LIN {X 0,Y 439.406,Z 545.749,A -85,B 0,C 180,E1 -8966.874,E2 -8966.874} C_VEL
LIN {X 0,Y 444.301,Z 559.149,A -85,B 0,C 180,E1 -8967.337,E2 -8967.337} C_VEL
LIN {X 0,Y 445.02,Z 561.087,A -85,B 0,C 180,E1 -8967.401,E2 -8967.401} C_VEL
LIN {X 0,Y 444.548,Z 605.152,A -85,B 0,C 180,E1 -8968.2,E2 -8968.2} C_VEL
LIN {X 0,Y 444.368,Z 618.583,A -85,B 0,C 180,E1 -8968.612,E2 -8968.612} C_VEL
LIN {X 0,Y 444.074,Z 631.835,A -85,B 0,C 180,E1 -8969.192,E2 -8969.192} C_VEL
LIN {X 0,Y 443.603,Z 644.701,A -85,B 0,C 180,E1 -8969.932,E2 -8969.932} C_VEL
LIN {X 0,Y 443.053,Z 657.633,A -85,B 0,C 180,E1 -8970.889,E2 -8970.889} C_VEL
LIN {X 0,Y 442.359,Z 670.207,A -85,B 0,C 180,E1 -8972.052,E2 -8972.052} C_VEL
LIN {X 0,Y 441.738,Z 680.558,A -85,B 0,C 180,E1 -8973.223,E2 -8973.223} C_VEL
LIN {X 0,Y 441.181,Z 690.099,A -85,B 0,C 180,E1 -8974.526,E2 -8974.526} C_VEL
LIN {X 0,Y 440.602,Z 699.018,A -85,B 0,C 180,E1 -8976,E2 -8976} C_VEL
LIN {X 0,Y 440.165,Z 706.273,A -85,B 0,C 180,E1 -8977.468,E2 -8977.468} C_VEL
LIN {X 0,Y 439.771,Z 712.189,A -85,B 0,C 180,E1 -8978.926,E2 -8978.926} C_VEL
LIN {X 0,Y 439.514,Z 717.633,A -85,B 0,C 180,E1 -8980.634,E2 -8980.634} C_VEL
LIN {X 0,Y 439.268,Z 721.644,A -85,B 0,C 180,E1 -8982.303,E2 -8982.303} C_VEL
LIN {X 0,Y 439.103,Z 724.753,A -85,B 0,C 180,E1 -8984.212,E2 -8984.212} C_VEL
LIN {X 0,Y 439.067,Z 726.387,A -85,B 0,C 180,E1 -8986.108,E2 -8986.108} C_VEL
LIN {X 0,Y 439.137,Z 726.572,A -85,B 0,C 180,E1 -8987.992,E2 -8987.992} C_VEL
LIN {X 0,Y 439.207,Z 725.332,A -85,B 0,C 180,E1 -8989.863,E2 -8989.863} C_VEL
LIN {X 0,Y 439.399,Z 722.692,A -85,B 0,C 180,E1 -8991.724,E2 -8991.724} C_VEL
LIN {X 0,Y 439.752,Z 718.586,A -85,B 0,C 180,E1 -8993.577,E2 -8993.577} C_VEL
LIN {X 0,Y 439.994,Z 714.453,A -85,B 0,C 180,E1 -8994.96,E2 -8994.96} C_VEL
LIN {X 0,Y 440.331,Z 709.35,A -85,B 0,C 180,E1 -8996.34,E2 -8996.34} C_VEL
LIN {X 0,Y 440.85,Z 701.986,A -85,B 0,C 180,E1 -8997.945,E2 -8997.945} C_VEL
LIN {X 0,Y 441.381,Z 694.239,A -85,B 0,C 180,E1 -8999.316,E2 -8999.316} C_VEL
LIN {X 0,Y 442.094,Z 684.837,A -85,B 0,C 180,E1 -9000.684,E2 -9000.684} C_VEL
LIN {X 0,Y 442.669,Z 674.365,A -85,B 0,C 180,E1 -9001.934,E2 -9001.934} C_VEL
LIN {X 0,Y 443.376,Z 662.58,A -85,B 0,C 180,E1 -9003.067,E2 -9003.067} C_VEL
LIN {X 0,Y 443.967,Z 650.958,A -85,B 0,C 180,E1 -9003.972,E2 -9003.972} C_VEL
LIN {X 0,Y 444.369,Z 638.23,A -85,B 0,C 180,E1 -9004.763,E2 -9004.763} C_VEL
LIN {X 0,Y 444.691,Z 624.706,A -85,B 0,C 180,E1 -9005.398,E2 -9005.398} C_VEL
LIN {X 0,Y 444.834,Z 611.284,A -85,B 0,C 180,E1 -9005.838,E2 -9005.838} C_VEL
LIN {X 0,Y 444.826,Z 592.596,A -85,B 0,C 180,E1 -9006.208,E2 -9006.208} C_VEL
LIN {X 0,Y 445.192,Z 560.426,A -85,B 0,C 180,E1 -9006.758,E2 -9006.758} C_VEL
LIN {X 0,Y 439.624,Z 545.984,A -85,B 0,C 180,E1 -9007.305,E2 -9007.305} C_VEL
LIN {X 0,Y 439.598,Z 545.729,A -85,B 0,C 180,E1 -9007.349,E2 -9007.349} C_VEL
LIN {X 0,Y 439.465,Z 545.745,A -85,B 0,C 180,E1 -9010.132,E2 -9010.132} C_VEL
LIN {X 0,Y 439.47,Z 545.745,A -85,B 0,C 180,E1 -9012.938,E2 -9012.938} C_VEL
LIN {X 0,Y 439.444,Z 545.746,A -85,B 0,C 180,E1 -9016.349,E2 -9016.349} C_VEL
LIN {X 0,Y 439.4,Z 545.753,A -85,B 0,C 180,E1 -9019.627,E2 -9019.627} C_VEL
LIN {X 0,Y 439.363,Z 545.754,A -85,B 0,C 180,E1 -9022.576,E2 -9022.576} C_VEL
LIN {X 0,Y 439.403,Z 545.75,A -85,B 0,C 180,E1 -9025.585,E2 -9025.585} C_VEL
LIN {X 0,Y 439.423,Z 545.743,A -85,B 0,C 180,E1 -9028.674,E2 -9028.674} C_VEL
LIN {X 0,Y 439.373,Z 545.747,A -85,B 0,C 180,E1 -9031.861,E2 -9031.861} C_VEL
LIN {X 0,Y 439.397,Z 545.747,A -85,B 0,C 180,E1 -9035.157,E2 -9035.157} C_VEL
LIN {X 0,Y 439.388,Z 545.749,A -85,B 0,C 180,E1 -9038.595,E2 -9038.595} C_VEL
LIN {X 0,Y 439.388,Z 545.754,A -85,B 0,C 180,E1 -9041.258,E2 -9041.258} C_VEL
LIN {X 0,Y 439.404,Z 545.749,A -85,B 0,C 180,E1 -9044.729,E2 -9044.729} C_VEL
LIN {X 0,Y 439.395,Z 545.748,A -85,B 0,C 180,E1 -9047.796,E2 -9047.796} C_VEL
LIN {X 0,Y 439.429,Z 545.745,A -85,B 0,C 180,E1 -9050.229,E2 -9050.229} C_VEL
LIN {X 0,Y 439.385,Z 545.756,A -85,B 0,C 180,E1 -9053.715,E2 -9053.715} C_VEL
LIN {X 0,Y 439.429,Z 545.847,A -85,B 0,C 180,E1 -9054.275,E2 -9054.275} C_VEL
LIN {X 0,Y 442.842,Z 561.566,A -85,B 0,C 180,E1 -9057.615,E2 -9057.615} C_VEL
LIN {X 0,Y 443.621,Z 565.787,A -85,B 0,C 180,E1 -9058.481,E2 -9058.481} C_VEL
LIN {X 0,Y 442.616,Z 582.035,A -85,B 0,C 180,E1 -9061.553,E2 -9061.553} C_VEL
LIN {X 0,Y 441.489,Z 601.988,A -85,B 0,C 180,E1 -9065.244,E2 -9065.244} C_VEL
LIN {X 0,Y 440.582,Z 621.12,A -85,B 0,C 180,E1 -9068.722,E2 -9068.722} C_VEL
LIN {X 0,Y 439.955,Z 635.532,A -85,B 0,C 180,E1 -9071.278,E2 -9071.278} C_VEL
LIN {X 0,Y 444.537,Z 670.934,A -85,B 0,C 180,E1 -9072.213,E2 -9072.213} C_VEL
LIN {X 0,Y 443.06,Z 749.107,A -85,B 0,C 180,E1 -9073.795,E2 -9073.795} C_VEL
LIN {X 0,Y 442.451,Z 763.207,A -85,B 0,C 180,E1 -9074.275,E2 -9074.275} C_VEL
LIN {X 0,Y 441.799,Z 775.931,A -85,B 0,C 180,E1 -9074.902,E2 -9074.902} C_VEL
LIN {X 0,Y 441.003,Z 788.207,A -85,B 0,C 180,E1 -9075.7,E2 -9075.7} C_VEL
LIN {X 0,Y 440.449,Z 799.159,A -85,B 0,C 180,E1 -9076.601,E2 -9076.601} C_VEL
LIN {X 0,Y 439.972,Z 809.643,A -85,B 0,C 180,E1 -9077.664,E2 -9077.664} C_VEL
LIN {X 0,Y 439.354,Z 819.768,A -85,B 0,C 180,E1 -9078.934,E2 -9078.934} C_VEL
LIN {X 0,Y 438.991,Z 828.76,A -85,B 0,C 180,E1 -9080.323,E2 -9080.323} C_VEL
LIN {X 0,Y 438.777,Z 835.975,A -85,B 0,C 180,E1 -9081.712,E2 -9081.712} C_VEL
LIN {X 0,Y 438.666,Z 842.745,A -85,B 0,C 180,E1 -9083.377,E2 -9083.377} C_VEL
LIN {X 0,Y 438.702,Z 847.553,A -85,B 0,C 180,E1 -9084.946,E2 -9084.946} C_VEL
LIN {X 0,Y 438.764,Z 850.593,A -85,B 0,C 180,E1 -9086.327,E2 -9086.327} C_VEL
LIN {X 0,Y 438.733,Z 852.033,A -85,B 0,C 180,E1 -9087.246,E2 -9087.246} C_VEL
LIN {X 0,Y 438.734,Z 853.013,A -85,B 0,C 180,E1 -9088.165,E2 -9088.165} C_VEL
LIN {X 0,Y 438.737,Z 853.57,A -85,B 0,C 180,E1 -9089.083,E2 -9089.083} C_VEL
LIN {X 0,Y 438.937,Z 853.735,A -85,B 0,C 180,E1 -9090.001,E2 -9090.001} C_VEL
LIN {X 0,Y 438.76,Z 853.392,A -85,B 0,C 180,E1 -9090.918,E2 -9090.918} C_VEL
LIN {X 0,Y 438.781,Z 852.625,A -85,B 0,C 180,E1 -9091.836,E2 -9091.836} C_VEL
LIN {X 0,Y 438.797,Z 851.434,A -85,B 0,C 180,E1 -9092.755,E2 -9092.755} C_VEL
LIN {X 0,Y 438.851,Z 848.799,A -85,B 0,C 180,E1 -9094.133,E2 -9094.133} C_VEL
LIN {X 0,Y 438.771,Z 845.065,A -85,B 0,C 180,E1 -9095.515,E2 -9095.515} C_VEL
LIN {X 0,Y 438.821,Z 840.059,A -85,B 0,C 180,E1 -9096.929,E2 -9096.929} C_VEL
LIN {X 0,Y 438.886,Z 833.994,A -85,B 0,C 180,E1 -9098.287,E2 -9098.287} C_VEL
LIN {X 0,Y 439.014,Z 826.334,A -85,B 0,C 180,E1 -9099.677,E2 -9099.677} C_VEL
LIN {X 0,Y 439.34,Z 816.842,A -85,B 0,C 180,E1 -9101.068,E2 -9101.068} C_VEL
LIN {X 0,Y 439.854,Z 806.195,A -85,B 0,C 180,E1 -9102.331,E2 -9102.331} C_VEL
LIN {X 0,Y 440.138,Z 798.182,A -85,B 0,C 180,E1 -9103.129,E2 -9103.129} C_VEL
LIN {X 0,Y 440.575,Z 788.32,A -85,B 0,C 180,E1 -9103.962,E2 -9103.962} C_VEL
LIN {X 0,Y 441.416,Z 774.803,A -85,B 0,C 180,E1 -9104.877,E2 -9104.877} C_VEL
LIN {X 0,Y 442.071,Z 761.506,A -85,B 0,C 180,E1 -9105.562,E2 -9105.562} C_VEL
LIN {X 0,Y 442.834,Z 747.018,A -85,B 0,C 180,E1 -9106.096,E2 -9106.096} C_VEL
LIN {X 0,Y 443.169,Z 732.682,A -85,B 0,C 180,E1 -9106.438,E2 -9106.438} C_VEL
LIN {X 0,Y 444.068,Z 670.071,A -85,B 0,C 180,E1 -9107.651,E2 -9107.651} C_VEL
LIN {X 0,Y 442.737,Z 654.934,A -85,B 0,C 180,E1 -9108.032,E2 -9108.032} C_VEL
LIN {X 0,Y 440.919,Z 632.046,A -85,B 0,C 180,E1 -9108.615,E2 -9108.615} C_VEL
LIN {X 0,Y 439.683,Z 620.875,A -85,B 0,C 180,E1 -9108.948,E2 -9108.948} C_VEL
LIN {X 0,Y 439.902,Z 603.534,A -85,B 0,C 180,E1 -9111.823,E2 -9111.823} C_VEL
LIN {X 0,Y 440.157,Z 584.473,A -85,B 0,C 180,E1 -9115.033,E2 -9115.033} C_VEL
LIN {X 0,Y 440.516,Z 566.826,A -85,B 0,C 180,E1 -9118.077,E2 -9118.077} C_VEL
LIN {X 0,Y 440.777,Z 553.487,A -85,B 0,C 180,E1 -9120.446,E2 -9120.446} C_VEL
LIN {X 0,Y 439.477,Z 545.744,A -85,B 0,C 180,E1 -9121.938,E2 -9121.938} C_VEL
LIN {X 0,Y 439.399,Z 545.752,A -85,B 0,C 180,E1 -9125.341,E2 -9125.341} C_VEL
LIN {X 0,Y 439.383,Z 545.753,A -85,B 0,C 180,E1 -9128.595,E2 -9128.595} C_VEL
LIN {X 0,Y 439.393,Z 545.752,A -85,B 0,C 180,E1 -9131.257,E2 -9131.257} C_VEL
LIN {X 0,Y 439.405,Z 545.752,A -85,B 0,C 180,E1 -9134.729,E2 -9134.729} C_VEL
LIN {X 0,Y 439.401,Z 545.749,A -85,B 0,C 180,E1 -9137.796,E2 -9137.796} C_VEL
LIN {X 0,Y 439.434,Z 545.747,A -85,B 0,C 180,E1 -9140.228,E2 -9140.228} C_VEL
LIN {X 0,Y 439.378,Z 545.752,A -85,B 0,C 180,E1 -9143.713,E2 -9143.713} C_VEL
LIN {X 0,Y 439.377,Z 545.755,A -85,B 0,C 180,E1 -9147.054,E2 -9147.054} C_VEL
LIN {X 0,Y 439.387,Z 545.754,A -85,B 0,C 180,E1 -9150.274,E2 -9150.274} C_VEL
LIN {X 0,Y 439.433,Z 545.749,A -85,B 0,C 180,E1 -9153.396,E2 -9153.396} C_VEL
LIN {X 0,Y 439.392,Z 545.758,A -85,B 0,C 180,E1 -9156.429,E2 -9156.429} C_VEL
LIN {X 0,Y 439.393,Z 545.753,A -85,B 0,C 180,E1 -9159.397,E2 -9159.397} C_VEL
LIN {X 0,Y 439.407,Z 545.753,A -85,B 0,C 180,E1 -9160.374,E2 -9160.374} C_VEL
LIN {X 0,Y 440.396,Z 548.536,A -85,B 0,C 180,E1 -9160.485,E2 -9160.485} C_VEL
LIN {X 0,Y 445.662,Z 561.095,A -85,B 0,C 180,E1 -9160.997,E2 -9160.997} C_VEL
LIN {X 0,Y 446.009,Z 561.957,A -85,B 0,C 180,E1 -9161.029,E2 -9161.029} C_VEL
LIN {X 0,Y 445.994,Z 595.08,A -85,B 0,C 180,E1 -9161.61,E2 -9161.61} C_VEL
LIN {X 0,Y 446.007,Z 609.272,A -85,B 0,C 180,E1 -9162.028,E2 -9162.028} C_VEL
LIN {X 0,Y 445.804,Z 623.559,A -85,B 0,C 180,E1 -9162.629,E2 -9162.629} C_VEL
LIN {X 0,Y 445.368,Z 637.072,A -85,B 0,C 180,E1 -9163.38,E2 -9163.38} C_VEL
LIN {X 0,Y 444.838,Z 650.124,A -85,B 0,C 180,E1 -9164.302,E2 -9164.302} C_VEL
LIN {X 0,Y 444.15,Z 663.194,A -85,B 0,C 180,E1 -9165.451,E2 -9165.451} C_VEL
LIN {X 0,Y 443.548,Z 673.013,A -85,B 0,C 180,E1 -9166.484,E2 -9166.484} C_VEL
LIN {X 0,Y 442.758,Z 683.962,A -85,B 0,C 180,E1 -9167.858,E2 -9167.858} C_VEL
LIN {X 0,Y 442.052,Z 693.037,A -85,B 0,C 180,E1 -9169.233,E2 -9169.233} C_VEL
LIN {X 0,Y 441.414,Z 701.82,A -85,B 0,C 180,E1 -9170.838,E2 -9170.838} C_VEL
LIN {X 0,Y 440.947,Z 708.047,A -85,B 0,C 180,E1 -9172.213,E2 -9172.213} C_VEL
LIN {X 0,Y 440.344,Z 713.376,A -85,B 0,C 180,E1 -9173.585,E2 -9173.585} C_VEL
LIN {X 0,Y 440.027,Z 719.004,A -85,B 0,C 180,E1 -9175.419,E2 -9175.419} C_VEL
LIN {X 0,Y 439.637,Z 723.262,A -85,B 0,C 180,E1 -9177.251,E2 -9177.251} C_VEL
LIN {X 0,Y 439.42,Z 726.213,A -85,B 0,C 180,E1 -9179.083,E2 -9179.083} C_VEL
LIN {X 0,Y 439.321,Z 727.927,A -85,B 0,C 180,E1 -9180.916,E2 -9180.916} C_VEL
LIN {X 0,Y 439.331,Z 728.446,A -85,B 0,C 180,E1 -9182.75,E2 -9182.75} C_VEL
LIN {X 0,Y 439.21,Z 727.821,A -85,B 0,C 180,E1 -9184.589,E2 -9184.589} C_VEL
LIN {X 0,Y 439.375,Z 725.987,A -85,B 0,C 180,E1 -9186.428,E2 -9186.428} C_VEL
LIN {X 0,Y 439.475,Z 722.948,A -85,B 0,C 180,E1 -9188.275,E2 -9188.275} C_VEL
LIN {X 0,Y 439.667,Z 718.609,A -85,B 0,C 180,E1 -9190.127,E2 -9190.127} C_VEL
LIN {X 0,Y 439.974,Z 712.852,A -85,B 0,C 180,E1 -9191.985,E2 -9191.985} C_VEL
LIN {X 0,Y 440.486,Z 705.487,A -85,B 0,C 180,E1 -9193.846,E2 -9193.846} C_VEL
LIN {X 0,Y 441.044,Z 697.51,A -85,B 0,C 180,E1 -9195.48,E2 -9195.48} C_VEL
LIN {X 0,Y 441.581,Z 689.227,A -85,B 0,C 180,E1 -9196.901,E2 -9196.901} C_VEL
LIN {X 0,Y 442.224,Z 679.63,A -85,B 0,C 180,E1 -9198.292,E2 -9198.292} C_VEL
LIN {X 0,Y 442.965,Z 667.969,A -85,B 0,C 180,E1 -9199.703,E2 -9199.703} C_VEL
LIN {X 0,Y 443.641,Z 656.875,A -85,B 0,C 180,E1 -9200.826,E2 -9200.826} C_VEL
LIN {X 0,Y 444.248,Z 645.173,A -85,B 0,C 180,E1 -9201.824,E2 -9201.824} C_VEL
LIN {X 0,Y 444.838,Z 631.595,A -85,B 0,C 180,E1 -9202.772,E2 -9202.772} C_VEL
LIN {X 0,Y 445.415,Z 616.975,A -85,B 0,C 180,E1 -9203.573,E2 -9203.573} C_VEL
LIN {X 0,Y 445.77,Z 601.844,A -85,B 0,C 180,E1 -9204.199,E2 -9204.199} C_VEL
LIN {X 0,Y 445.907,Z 586.802,A -85,B 0,C 180,E1 -9204.635,E2 -9204.635} C_VEL
LIN {X 0,Y 445.984,Z 563.306,A -85,B 0,C 180,E1 -9205.079,E2 -9205.079} C_VEL
LIN {X 0,Y 439.464,Z 545.989,A -85,B 0,C 180,E1 -9205.687,E2 -9205.687} C_VEL
LIN {X 0,Y 439.43,Z 545.751,A -85,B 0,C 180,E1 -9205.837,E2 -9205.837} C_VEL
LIN {X 0,Y 439.419,Z 545.747,A -85,B 0,C 180,E1 -9208.673,E2 -9208.673} C_VEL
LIN {X 0,Y 439.372,Z 545.758,A -85,B 0,C 180,E1 -9212.03,E2 -9212.03} C_VEL
LIN {X 0,Y 439.395,Z 545.747,A -85,B 0,C 180,E1 -9215.34,E2 -9215.34} C_VEL
LIN {X 0,Y 439.379,Z 545.752,A -85,B 0,C 180,E1 -9218.595,E2 -9218.595} C_VEL
LIN {X 0,Y 439.389,Z 545.748,A -85,B 0,C 180,E1 -9221.256,E2 -9221.256} C_VEL
LIN {X 0,Y 439.4,Z 545.749,A -85,B 0,C 180,E1 -9224.729,E2 -9224.729} C_VEL
LIN {X 0,Y 439.396,Z 545.749,A -85,B 0,C 180,E1 -9227.795,E2 -9227.795} C_VEL
LIN {X 0,Y 439.436,Z 545.748,A -85,B 0,C 180,E1 -9230.228,E2 -9230.228} C_VEL
LIN {X 0,Y 439.376,Z 545.75,A -85,B 0,C 180,E1 -9233.712,E2 -9233.712} C_VEL
LIN {X 0,Y 439.372,Z 545.752,A -85,B 0,C 180,E1 -9237.053,E2 -9237.053} C_VEL
LIN {X 0,Y 439.382,Z 545.753,A -85,B 0,C 180,E1 -9240.274,E2 -9240.274} C_VEL
LIN {X 0,Y 439.429,Z 545.743,A -85,B 0,C 180,E1 -9243.396,E2 -9243.396} C_VEL
LIN {X 0,Y 439.387,Z 545.753,A -85,B 0,C 180,E1 -9246.429,E2 -9246.429} C_VEL
LIN {X 0,Y 439.388,Z 545.749,A -85,B 0,C 180,E1 -9249.397,E2 -9249.397} C_VEL
LIN {X 0,Y 439.43,Z 545.745,A -85,B 0,C 180,E1 -9252.309,E2 -9252.309} C_VEL
LIN {X 0,Y 439.447,Z 545.745,A -85,B 0,C 180,E1 -9255.173,E2 -9255.173} C_VEL
LIN {X 0,Y 439.482,Z 545.736,A -85,B 0,C 180,E1 -9258.001,E2 -9258.001} C_VEL
LIN {X 0,Y 439.528,Z 545.731,A -85,B 0,C 180,E1 -9261.547,E2 -9261.547} C_VEL
LIN {X 0,Y 438.908,Z 545.81,A -85,B 0,C 180,E1 -9262.313,E2 -9262.313} C_VEL
LIN {X 0,Y 436.034,Z 546.171,A -85,B 0,C 180,E1 -9263.556,E2 -9263.556} C_VEL
LIN {X 0,Y 433.558,Z 546.481,A -85,B 0,C 180,E1 -9264.559,E2 -9264.559} C_VEL
LIN {X 0,Y 432.477,Z 546.614,A -85,B 0,C 180,E1 -9265.334,E2 -9265.334} C_VEL
LIN {X 0,Y 432.382,Z 546.622,A -85,B 0,C 180,E1 -9265.597,E2 -9265.597} C_VEL
LIN {X 0,Y 432.604,Z 546.593,A -85,B 0,C 180,E1 -9268.137,E2 -9268.137} C_VEL
LIN {X 0,Y 432.732,Z 546.577,A -85,B 0,C 180,E1 -9269.999,E2 -9269.999} C_VEL
LIN {X 0,Y 432.604,Z 546.596,A -85,B 0,C 180,E1 -9272.793,E2 -9272.793} C_VEL
LIN {X 0,Y 432.562,Z 546.599,A -85,B 0,C 180,E1 -9276.53,E2 -9276.53} C_VEL
LIN {X 0,Y 432.441,Z 546.621,A -85,B 0,C 180,E1 -9279.353,E2 -9279.353} C_VEL
LIN {X 0,Y 432.442,Z 546.615,A -85,B 0,C 180,E1 -9282.812,E2 -9282.812} C_VEL
LIN {X 0,Y 432.409,Z 546.617,A -85,B 0,C 180,E1 -9286.479,E2 -9286.479} C_VEL
LIN {X 0,Y 432.335,Z 546.629,A -85,B 0,C 180,E1 -9289.96,E2 -9289.96} C_VEL
LIN {X 0,Y 432.316,Z 546.63,A -85,B 0,C 180,E1 -9292.964,E2 -9292.964} C_VEL
LIN {X 0,Y 432.361,Z 546.626,A -85,B 0,C 180,E1 -9296.032,E2 -9296.032} C_VEL
LIN {X 0,Y 432.348,Z 546.627,A -85,B 0,C 180,E1 -9299.186,E2 -9299.186} C_VEL
LIN {X 0,Y 432.327,Z 546.629,A -85,B 0,C 180,E1 -9302.294,E2 -9302.294} C_VEL
LIN {X 0,Y 432.336,Z 546.627,A -85,B 0,C 180,E1 -9304.677,E2 -9304.677} C_VEL
LIN {X 0,Y 432.346,Z 546.629,A -85,B 0,C 180,E1 -9308.148,E2 -9308.148} C_VEL
LIN {X 0,Y 432.361,Z 546.627,A -85,B 0,C 180,E1 -9311.607,E2 -9311.607} C_VEL
LIN {X 0,Y 432.332,Z 546.63,A -85,B 0,C 180,E1 -9314.347,E2 -9314.347} C_VEL
LIN {X 0,Y 432.36,Z 546.623,A -85,B 0,C 180,E1 -9317.009,E2 -9317.009} C_VEL
LIN {X 0,Y 432.355,Z 546.629,A -85,B 0,C 180,E1 -9319.816,E2 -9319.816} C_VEL
LIN {X 0,Y 432.312,Z 546.629,A -85,B 0,C 180,E1 -9323.023,E2 -9323.023} C_VEL
LIN {X 0,Y 432.371,Z 546.626,A -85,B 0,C 180,E1 -9326.535,E2 -9326.535} C_VEL
LIN {X 0,Y 432.415,Z 546.866,A -85,B 0,C 180,E1 -9326.623,E2 -9326.623} C_VEL
LIN {X 0,Y 438.178,Z 562.466,A -85,B 0,C 180,E1 -9327.152,E2 -9327.152} C_VEL
LIN {X 0,Y 437.739,Z 605.294,A -85,B 0,C 180,E1 -9327.943,E2 -9327.943} C_VEL
LIN {X 0,Y 437.568,Z 619.263,A -85,B 0,C 180,E1 -9328.372,E2 -9328.372} C_VEL
LIN {X 0,Y 437.269,Z 632.342,A -85,B 0,C 180,E1 -9328.948,E2 -9328.948} C_VEL
LIN {X 0,Y 436.792,Z 645.03,A -85,B 0,C 180,E1 -9329.681,E2 -9329.681} C_VEL
LIN {X 0,Y 436.274,Z 657.064,A -85,B 0,C 180,E1 -9330.562,E2 -9330.562} C_VEL
LIN {X 0,Y 435.648,Z 668.401,A -85,B 0,C 180,E1 -9331.582,E2 -9331.582} C_VEL
LIN {X 0,Y 434.942,Z 679.636,A -85,B 0,C 180,E1 -9332.821,E2 -9332.821} C_VEL
LIN {X 0,Y 434.319,Z 689.176,A -85,B 0,C 180,E1 -9334.094,E2 -9334.094} C_VEL
LIN {X 0,Y 433.754,Z 698.457,A -85,B 0,C 180,E1 -9335.596,E2 -9335.596} C_VEL
LIN {X 0,Y 433.257,Z 706.021,A -85,B 0,C 180,E1 -9337.089,E2 -9337.089} C_VEL
LIN {X 0,Y 432.845,Z 712.177,A -85,B 0,C 180,E1 -9338.573,E2 -9338.573} C_VEL
LIN {X 0,Y 432.568,Z 717.133,A -85,B 0,C 180,E1 -9340.051,E2 -9340.051} C_VEL
LIN {X 0,Y 432.356,Z 721.035,A -85,B 0,C 180,E1 -9341.52,E2 -9341.52} C_VEL
LIN {X 0,Y 432.158,Z 723.999,A -85,B 0,C 180,E1 -9342.979,E2 -9342.979} C_VEL
LIN {X 0,Y 432.037,Z 726.542,A -85,B 0,C 180,E1 -9344.914,E2 -9344.914} C_VEL
LIN {X 0,Y 432.078,Z 727.631,A -85,B 0,C 180,E1 -9346.838,E2 -9346.838} C_VEL
LIN {X 0,Y 432.111,Z 727.328,A -85,B 0,C 180,E1 -9348.746,E2 -9348.746} C_VEL
LIN {X 0,Y 432.279,Z 725.572,A -85,B 0,C 180,E1 -9350.644,E2 -9350.644} C_VEL
LIN {X 0,Y 432.549,Z 722.374,A -85,B 0,C 180,E1 -9352.532,E2 -9352.532} C_VEL
LIN {X 0,Y 432.895,Z 717.686,A -85,B 0,C 180,E1 -9354.41,E2 -9354.41} C_VEL
LIN {X 0,Y 433.213,Z 713.068,A -85,B 0,C 180,E1 -9355.814,E2 -9355.814} C_VEL
LIN {X 0,Y 433.767,Z 706.35,A -85,B 0,C 180,E1 -9357.447,E2 -9357.447} C_VEL
LIN {X 0,Y 434.253,Z 699.278,A -85,B 0,C 180,E1 -9358.841,E2 -9358.841} C_VEL
LIN {X 0,Y 434.957,Z 690.7,A -85,B 0,C 180,E1 -9360.232,E2 -9360.232} C_VEL
LIN {X 0,Y 435.498,Z 682.189,A -85,B 0,C 180,E1 -9361.387,E2 -9361.387} C_VEL
LIN {X 0,Y 436.155,Z 672.098,A -85,B 0,C 180,E1 -9362.53,E2 -9362.53} C_VEL
LIN {X 0,Y 436.802,Z 660.849,A -85,B 0,C 180,E1 -9363.575,E2 -9363.575} C_VEL
LIN {X 0,Y 437.413,Z 648.462,A -85,B 0,C 180,E1 -9364.493,E2 -9364.493} C_VEL
LIN {X 0,Y 437.802,Z 635.629,A -85,B 0,C 180,E1 -9365.239,E2 -9365.239} C_VEL
LIN {X 0,Y 438.099,Z 621.765,A -85,B 0,C 180,E1 -9365.836,E2 -9365.836} C_VEL
LIN {X 0,Y 438.132,Z 608.616,A -85,B 0,C 180,E1 -9366.225,E2 -9366.225} C_VEL
LIN {X 0,Y 438.569,Z 562.004,A -85,B 0,C 180,E1 -9367.058,E2 -9367.058} C_VEL
LIN {X 0,Y 432.674,Z 547.122,A -85,B 0,C 180,E1 -9367.662,E2 -9367.662} C_VEL
LIN {X 0,Y 432.56,Z 546.606,A -85,B 0,C 180,E1 -9367.698,E2 -9367.698} C_VEL
LIN {X 0,Y 432.405,Z 546.625,A -85,B 0,C 180,E1 -9371.247,E2 -9371.247} C_VEL
LIN {X 0,Y 432.428,Z 546.624,A -85,B 0,C 180,E1 -9373.152,E2 -9373.152} C_VEL
LIN {X 0,Y 432.409,Z 546.622,A -85,B 0,C 180,E1 -9376.48,E2 -9376.48} C_VEL
LIN {X 0,Y 432.336,Z 546.633,A -85,B 0,C 180,E1 -9379.961,E2 -9379.961} C_VEL
LIN {X 0,Y 432.317,Z 546.634,A -85,B 0,C 180,E1 -9382.965,E2 -9382.965} C_VEL
LIN {X 0,Y 432.362,Z 546.625,A -85,B 0,C 180,E1 -9386.033,E2 -9386.033} C_VEL
LIN {X 0,Y 432.35,Z 546.629,A -85,B 0,C 180,E1 -9389.187,E2 -9389.187} C_VEL
LIN {X 0,Y 432.323,Z 546.623,A -85,B 0,C 180,E1 -9392.294,E2 -9392.294} C_VEL
LIN {X 0,Y 432.338,Z 546.624,A -85,B 0,C 180,E1 -9394.678,E2 -9394.678} C_VEL
LIN {X 0,Y 432.345,Z 546.626,A -85,B 0,C 180,E1 -9398.15,E2 -9398.15} C_VEL
LIN {X 0,Y 432.333,Z 546.629,A -85,B 0,C 180,E1 -9401.603,E2 -9401.603} C_VEL
LIN {X 0,Y 432.339,Z 546.627,A -85,B 0,C 180,E1 -9404.347,E2 -9404.347} C_VEL
LIN {X 0,Y 432.319,Z 546.635,A -85,B 0,C 180,E1 -9407.016,E2 -9407.016} C_VEL
LIN {X 0,Y 432.336,Z 546.63,A -85,B 0,C 180,E1 -9409.821,E2 -9409.821} C_VEL
LIN {X 0,Y 432.315,Z 546.639,A -85,B 0,C 180,E1 -9413.024,E2 -9413.024} C_VEL
LIN {X 0,Y 432.36,Z 546.675,A -85,B 0,C 180,E1 -9414.006,E2 -9414.006} C_VEL
LIN {X 0,Y 435.767,Z 562.166,A -85,B 0,C 180,E1 -9417.361,E2 -9417.361} C_VEL
LIN {X 0,Y 436.683,Z 567.856,A -85,B 0,C 180,E1 -9418.539,E2 -9418.539} C_VEL
LIN {X 0,Y 435.502,Z 585.024,A -85,B 0,C 180,E1 -9421.835,E2 -9421.835} C_VEL
LIN {X 0,Y 434.382,Z 603.876,A -85,B 0,C 180,E1 -9425.38,E2 -9425.38} C_VEL
LIN {X 0,Y 433.482,Z 622.667,A -85,B 0,C 180,E1 -9428.855,E2 -9428.855} C_VEL
LIN {X 0,Y 432.98,Z 633.899,A -85,B 0,C 180,E1 -9430.918,E2 -9430.918} C_VEL
LIN {X 0,Y 437.731,Z 671.401,A -85,B 0,C 180,E1 -9431.951,E2 -9431.951} C_VEL
LIN {X 0,Y 436.195,Z 747.525,A -85,B 0,C 180,E1 -9433.533,E2 -9433.533} C_VEL
LIN {X 0,Y 435.651,Z 761.005,A -85,B 0,C 180,E1 -9433.993,E2 -9433.993} C_VEL
LIN {X 0,Y 434.921,Z 773.533,A -85,B 0,C 180,E1 -9434.597,E2 -9434.597} C_VEL
LIN {X 0,Y 434.169,Z 785.308,A -85,B 0,C 180,E1 -9435.35,E2 -9435.35} C_VEL
LIN {X 0,Y 433.517,Z 796.817,A -85,B 0,C 180,E1 -9436.286,E2 -9436.286} C_VEL
LIN {X 0,Y 433.016,Z 807.345,A -85,B 0,C 180,E1 -9437.344,E2 -9437.344} C_VEL
LIN {X 0,Y 432.452,Z 816.921,A -85,B 0,C 180,E1 -9438.517,E2 -9438.517} C_VEL
LIN {X 0,Y 431.963,Z 826.214,A -85,B 0,C 180,E1 -9439.928,E2 -9439.928} C_VEL
LIN {X 0,Y 431.752,Z 833.758,A -85,B 0,C 180,E1 -9441.341,E2 -9441.341} C_VEL
LIN {X 0,Y 431.626,Z 838.874,A -85,B 0,C 180,E1 -9442.516,E2 -9442.516} C_VEL
LIN {X 0,Y 431.646,Z 843.843,A -85,B 0,C 180,E1 -9443.925,E2 -9443.925} C_VEL
LIN {X 0,Y 431.688,Z 847.634,A -85,B 0,C 180,E1 -9445.331,E2 -9445.331} C_VEL
LIN {X 0,Y 431.726,Z 849.569,A -85,B 0,C 180,E1 -9446.267,E2 -9446.267} C_VEL
LIN {X 0,Y 431.692,Z 851.024,A -85,B 0,C 180,E1 -9447.201,E2 -9447.201} C_VEL
LIN {X 0,Y 431.697,Z 852.008,A -85,B 0,C 180,E1 -9448.135,E2 -9448.135} C_VEL
LIN {X 0,Y 431.706,Z 852.566,A -85,B 0,C 180,E1 -9449.068,E2 -9449.068} C_VEL
LIN {X 0,Y 431.916,Z 852.729,A -85,B 0,C 180,E1 -9450.001,E2 -9450.001} C_VEL
LIN {X 0,Y 431.729,Z 852.388,A -85,B 0,C 180,E1 -9450.933,E2 -9450.933} C_VEL
LIN {X 0,Y 431.745,Z 851.613,A -85,B 0,C 180,E1 -9451.866,E2 -9451.866} C_VEL
LIN {X 0,Y 431.756,Z 850.407,A -85,B 0,C 180,E1 -9452.8,E2 -9452.8} C_VEL
LIN {X 0,Y 431.811,Z 847.757,A -85,B 0,C 180,E1 -9454.201,E2 -9454.201} C_VEL
LIN {X 0,Y 431.709,Z 844.008,A -85,B 0,C 180,E1 -9455.606,E2 -9455.606} C_VEL
LIN {X 0,Y 431.735,Z 838.587,A -85,B 0,C 180,E1 -9457.143,E2 -9457.143} C_VEL
LIN {X 0,Y 431.815,Z 831.739,A -85,B 0,C 180,E1 -9458.659,E2 -9458.659} C_VEL
LIN {X 0,Y 431.976,Z 823.755,A -85,B 0,C 180,E1 -9460.073,E2 -9460.073} C_VEL
LIN {X 0,Y 432.381,Z 813.918,A -85,B 0,C 180,E1 -9461.486,E2 -9461.486} C_VEL
LIN {X 0,Y 432.795,Z 804.602,A -85,B 0,C 180,E1 -9462.586,E2 -9462.586} C_VEL
LIN {X 0,Y 433.253,Z 795.935,A -85,B 0,C 180,E1 -9463.449,E2 -9463.449} C_VEL
LIN {X 0,Y 433.856,Z 784.218,A -85,B 0,C 180,E1 -9464.422,E2 -9464.422} C_VEL
LIN {X 0,Y 434.694,Z 771.9,A -85,B 0,C 180,E1 -9465.232,E2 -9465.232} C_VEL
LIN {X 0,Y 435.305,Z 759.462,A -85,B 0,C 180,E1 -9465.871,E2 -9465.871} C_VEL
LIN {X 0,Y 436.051,Z 744.898,A -85,B 0,C 180,E1 -9466.413,E2 -9466.413} C_VEL
LIN {X 0,Y 436.408,Z 728.983,A -85,B 0,C 180,E1 -9466.791,E2 -9466.791} C_VEL
LIN {X 0,Y 437.377,Z 670.558,A -85,B 0,C 180,E1 -9467.958,E2 -9467.958} C_VEL
LIN {X 0,Y 436.092,Z 655.625,A -85,B 0,C 180,E1 -9468.347,E2 -9468.347} C_VEL
LIN {X 0,Y 434.31,Z 632.621,A -85,B 0,C 180,E1 -9468.959,E2 -9468.959} C_VEL
LIN {X 0,Y 432.65,Z 618.215,A -85,B 0,C 180,E1 -9469.401,E2 -9469.401} C_VEL
LIN {X 0,Y 432.873,Z 599.658,A -85,B 0,C 180,E1 -9472.546,E2 -9472.546} C_VEL
LIN {X 0,Y 433.185,Z 581.259,A -85,B 0,C 180,E1 -9475.722,E2 -9475.722} C_VEL
LIN {X 0,Y 433.688,Z 560.796,A -85,B 0,C 180,E1 -9479.355,E2 -9479.355} C_VEL
LIN {X 0,Y 433.778,Z 554.802,A -85,B 0,C 180,E1 -9480.454,E2 -9480.454} C_VEL
LIN {X 0,Y 432.415,Z 546.624,A -85,B 0,C 180,E1 -9482.068,E2 -9482.068} C_VEL
LIN {X 0,Y 432.349,Z 546.628,A -85,B 0,C 180,E1 -9485.632,E2 -9485.632} C_VEL
LIN {X 0,Y 432.351,Z 546.628,A -85,B 0,C 180,E1 -9489.343,E2 -9489.343} C_VEL
LIN {X 0,Y 432.338,Z 546.628,A -85,B 0,C 180,E1 -9491.797,E2 -9491.797} C_VEL
LIN {X 0,Y 432.338,Z 546.63,A -85,B 0,C 180,E1 -9494.347,E2 -9494.347} C_VEL
LIN {X 0,Y 432.325,Z 546.635,A -85,B 0,C 180,E1 -9497.016,E2 -9497.016} C_VEL
LIN {X 0,Y 432.341,Z 546.629,A -85,B 0,C 180,E1 -9499.82,E2 -9499.82} C_VEL
LIN {X 0,Y 432.311,Z 546.636,A -85,B 0,C 180,E1 -9503.022,E2 -9503.022} C_VEL
LIN {X 0,Y 432.364,Z 546.628,A -85,B 0,C 180,E1 -9505.996,E2 -9505.996} C_VEL
LIN {X 0,Y 432.352,Z 546.627,A -85,B 0,C 180,E1 -9509.489,E2 -9509.489} C_VEL
LIN {X 0,Y 432.396,Z 546.627,A -85,B 0,C 180,E1 -9512.928,E2 -9512.928} C_VEL
LIN {X 0,Y 432.376,Z 546.629,A -85,B 0,C 180,E1 -9516.023,E2 -9516.023} C_VEL
LIN {X 0,Y 432.357,Z 546.63,A -85,B 0,C 180,E1 -9519.544,E2 -9519.544} C_VEL
LIN {X 0,Y 432.341,Z 546.633,A -85,B 0,C 180,E1 -9519.977,E2 -9519.977} C_VEL
LIN {X 0,Y 433.33,Z 549.439,A -85,B 0,C 180,E1 -9520.091,E2 -9520.091} C_VEL
LIN {X 0,Y 439.056,Z 562.513,A -85,B 0,C 180,E1 -9520.655,E2 -9520.655} C_VEL
LIN {X 0,Y 439.535,Z 563.956,A -85,B 0,C 180,E1 -9520.707,E2 -9520.707} C_VEL
LIN {X 0,Y 439.409,Z 596.448,A -85,B 0,C 180,E1 -9521.291,E2 -9521.291} C_VEL
LIN {X 0,Y 439.404,Z 611.1,A -85,B 0,C 180,E1 -9521.734,E2 -9521.734} C_VEL
LIN {X 0,Y 439.194,Z 625.557,A -85,B 0,C 180,E1 -9522.359,E2 -9522.359} C_VEL
LIN {X 0,Y 438.751,Z 638.963,A -85,B 0,C 180,E1 -9523.122,E2 -9523.122} C_VEL
LIN {X 0,Y 438.204,Z 651.934,A -85,B 0,C 180,E1 -9524.058,E2 -9524.058} C_VEL
LIN {X 0,Y 437.555,Z 663.782,A -85,B 0,C 180,E1 -9525.108,E2 -9525.108} C_VEL
LIN {X 0,Y 436.846,Z 674.656,A -85,B 0,C 180,E1 -9526.272,E2 -9526.272} C_VEL
LIN {X 0,Y 435.978,Z 685.499,A -85,B 0,C 180,E1 -9527.667,E2 -9527.667} C_VEL
LIN {X 0,Y 435.247,Z 694.531,A -85,B 0,C 180,E1 -9529.063,E2 -9529.063} C_VEL
LIN {X 0,Y 434.56,Z 703.278,A -85,B 0,C 180,E1 -9530.692,E2 -9530.692} C_VEL
LIN {X 0,Y 434.069,Z 709.459,A -85,B 0,C 180,E1 -9532.089,E2 -9532.089} C_VEL
LIN {X 0,Y 433.422,Z 714.745,A -85,B 0,C 180,E1 -9533.482,E2 -9533.482} C_VEL
LIN {X 0,Y 433.075,Z 720.304,A -85,B 0,C 180,E1 -9535.345,E2 -9535.345} C_VEL
LIN {X 0,Y 432.673,Z 724.489,A -85,B 0,C 180,E1 -9537.206,E2 -9537.206} C_VEL
LIN {X 0,Y 432.43,Z 727.38,A -85,B 0,C 180,E1 -9539.068,E2 -9539.068} C_VEL
LIN {X 0,Y 432.309,Z 729.052,A -85,B 0,C 180,E1 -9540.931,E2 -9540.931} C_VEL
LIN {X 0,Y 432.311,Z 729.511,A -85,B 0,C 180,E1 -9542.795,E2 -9542.795} C_VEL
LIN {X 0,Y 432.194,Z 728.811,A -85,B 0,C 180,E1 -9544.663,E2 -9544.663} C_VEL
LIN {X 0,Y 432.368,Z 726.896,A -85,B 0,C 180,E1 -9546.533,E2 -9546.533} C_VEL
LIN {X 0,Y 432.477,Z 723.77,A -85,B 0,C 180,E1 -9548.41,E2 -9548.41} C_VEL
LIN {X 0,Y 432.684,Z 719.333,A -85,B 0,C 180,E1 -9550.292,E2 -9550.292} C_VEL
LIN {X 0,Y 433.021,Z 713.464,A -85,B 0,C 180,E1 -9552.18,E2 -9552.18} C_VEL
LIN {X 0,Y 433.492,Z 707,A -85,B 0,C 180,E1 -9553.835,E2 -9553.835} C_VEL
LIN {X 0,Y 434.044,Z 699.11,A -85,B 0,C 180,E1 -9555.495,E2 -9555.495} C_VEL
LIN {X 0,Y 434.709,Z 689.694,A -85,B 0,C 180,E1 -9557.132,E2 -9557.132} C_VEL
LIN {X 0,Y 435.368,Z 679.637,A -85,B 0,C 180,E1 -9558.591,E2 -9558.591} C_VEL
LIN {X 0,Y 436.128,Z 667.748,A -85,B 0,C 180,E1 -9560.025,E2 -9560.025} C_VEL
LIN {X 0,Y 436.911,Z 655.017,A -85,B 0,C 180,E1 -9561.291,E2 -9561.291} C_VEL
LIN {X 0,Y 437.605,Z 642.729,A -85,B 0,C 180,E1 -9562.297,E2 -9562.297} C_VEL
LIN {X 0,Y 438.109,Z 630.248,A -85,B 0,C 180,E1 -9563.142,E2 -9563.142} C_VEL
LIN {X 0,Y 438.691,Z 615.822,A -85,B 0,C 180,E1 -9563.912,E2 -9563.912} C_VEL
LIN {X 0,Y 439.036,Z 600.636,A -85,B 0,C 180,E1 -9564.522,E2 -9564.522} C_VEL
LIN {X 0,Y 439.142,Z 586.078,A -85,B 0,C 180,E1 -9564.927,E2 -9564.927} C_VEL
LIN {X 0,Y 439.22,Z 564.913,A -85,B 0,C 180,E1 -9565.335,E2 -9565.335} C_VEL
LIN {X 0,Y 432.421,Z 546.794,A -85,B 0,C 180,E1 -9565.975,E2 -9565.975} C_VEL
LIN {X 0,Y 432.344,Z 546.628,A -85,B 0,C 180,E1 -9569.187,E2 -9569.187} C_VEL
LIN {X 0,Y 432.324,Z 546.631,A -85,B 0,C 180,E1 -9572.442,E2 -9572.442} C_VEL
LIN {X 0,Y 432.345,Z 546.627,A -85,B 0,C 180,E1 -9575.631,E2 -9575.631} C_VEL
LIN {X 0,Y 432.347,Z 546.625,A -85,B 0,C 180,E1 -9579.343,E2 -9579.343} C_VEL
LIN {X 0,Y 432.333,Z 546.629,A -85,B 0,C 180,E1 -9581.796,E2 -9581.796} C_VEL
LIN {X 0,Y 432.333,Z 546.635,A -85,B 0,C 180,E1 -9584.347,E2 -9584.347} C_VEL
LIN {X 0,Y 432.32,Z 546.629,A -85,B 0,C 180,E1 -9587.015,E2 -9587.015} C_VEL
LIN {X 0,Y 432.341,Z 546.627,A -85,B 0,C 180,E1 -9589.819,E2 -9589.819} C_VEL
LIN {X 0,Y 432.314,Z 546.631,A -85,B 0,C 180,E1 -9593.022,E2 -9593.022} C_VEL
LIN {X 0,Y 432.359,Z 546.626,A -85,B 0,C 180,E1 -9595.996,E2 -9595.996} C_VEL
LIN {X 0,Y 432.347,Z 546.625,A -85,B 0,C 180,E1 -9599.489,E2 -9599.489} C_VEL
LIN {X 0,Y 432.391,Z 546.624,A -85,B 0,C 180,E1 -9602.928,E2 -9602.928} C_VEL
LIN {X 0,Y 432.371,Z 546.623,A -85,B 0,C 180,E1 -9606.023,E2 -9606.023} C_VEL
LIN {X 0,Y 432.349,Z 546.629,A -85,B 0,C 180,E1 -9609.046,E2 -9609.046} C_VEL
LIN {X 0,Y 432.377,Z 546.622,A -85,B 0,C 180,E1 -9612.011,E2 -9612.011} C_VEL
LIN {X 0,Y 432.395,Z 546.627,A -85,B 0,C 180,E1 -9614.926,E2 -9614.926} C_VEL
LIN {X 0,Y 432.458,Z 546.611,A -85,B 0,C 180,E1 -9617.803,E2 -9617.803} C_VEL
LIN {X 0,Y 432.49,Z 546.609,A -85,B 0,C 180,E1 -9621.59,E2 -9621.59} C_VEL
LIN {X 0,Y 432.596,Z 546.595,A -85,B 0,C 180,E1 -9624.406,E2 -9624.406} C_VEL
LIN {X 0,Y 432.382,Z 546.622,A -85,B 0,C 180,E1 -9625.597,E2 -9625.597} C_VEL
LIN {X 0,Y 431.702,Z 546.707,A -85,B 0,C 180,E1 -9626.376,E2 -9626.376} C_VEL
LIN {X 0,Y 428.889,Z 547.058,A -85,B 0,C 180,E1 -9627.643,E2 -9627.643} C_VEL
LIN {X 0,Y 426.582,Z 547.346,A -85,B 0,C 180,E1 -9628.666,E2 -9628.666} C_VEL
LIN {X 0,Y 425.673,Z 547.461,A -85,B 0,C 180,E1 -9629.456,E2 -9629.456} C_VEL
LIN {X 0,Y 425.642,Z 547.461,A -85,B 0,C 180,E1 -9629.722,E2 -9629.722} C_VEL
LIN {X 0,Y 425.556,Z 547.475,A -85,B 0,C 180,E1 -9632.839,E2 -9632.839} C_VEL
LIN {X 0,Y 425.52,Z 547.477,A -85,B 0,C 180,E1 -9636.638,E2 -9636.638} C_VEL
LIN {X 0,Y 425.4,Z 547.496,A -85,B 0,C 180,E1 -9639.509,E2 -9639.509} C_VEL
LIN {X 0,Y 425.401,Z 547.493,A -85,B 0,C 180,E1 -9642.91,E2 -9642.91} C_VEL
LIN {X 0,Y 425.358,Z 547.496,A -85,B 0,C 180,E1 -9646.605,E2 -9646.605} C_VEL
LIN {X 0,Y 425.325,Z 547.506,A -85,B 0,C 180,E1 -9649.635,E2 -9649.635} C_VEL
LIN {X 0,Y 425.303,Z 547.508,A -85,B 0,C 180,E1 -9653.365,E2 -9653.365} C_VEL
LIN {X 0,Y 425.344,Z 547.498,A -85,B 0,C 180,E1 -9656.844,E2 -9656.844} C_VEL
LIN {X 0,Y 425.314,Z 547.509,A -85,B 0,C 180,E1 -9659.717,E2 -9659.717} C_VEL
LIN {X 0,Y 425.279,Z 547.506,A -85,B 0,C 180,E1 -9663.047,E2 -9663.047} C_VEL
LIN {X 0,Y 425.28,Z 547.512,A -85,B 0,C 180,E1 -9665.929,E2 -9665.929} C_VEL
LIN {X 0,Y 425.305,Z 547.503,A -85,B 0,C 180,E1 -9669.045,E2 -9669.045} C_VEL
LIN {X 0,Y 425.31,Z 547.509,A -85,B 0,C 180,E1 -9671.962,E2 -9671.962} C_VEL
LIN {X 0,Y 425.308,Z 547.503,A -85,B 0,C 180,E1 -9675.279,E2 -9675.279} C_VEL
LIN {X 0,Y 425.305,Z 547.504,A -85,B 0,C 180,E1 -9678.626,E2 -9678.626} C_VEL
LIN {X 0,Y 425.321,Z 547.5,A -85,B 0,C 180,E1 -9681.104,E2 -9681.104} C_VEL
LIN {X 0,Y 425.295,Z 547.505,A -85,B 0,C 180,E1 -9684.664,E2 -9684.664} C_VEL
LIN {X 0,Y 425.33,Z 547.504,A -85,B 0,C 180,E1 -9686.324,E2 -9686.324} C_VEL
LIN {X 0,Y 431.437,Z 564.273,A -85,B 0,C 180,E1 -9686.91,E2 -9686.91} C_VEL
LIN {X 0,Y 430.943,Z 606.17,A -85,B 0,C 180,E1 -9687.699,E2 -9687.699} C_VEL
LIN {X 0,Y 430.772,Z 620.111,A -85,B 0,C 180,E1 -9688.133,E2 -9688.133} C_VEL
LIN {X 0,Y 430.396,Z 634.337,A -85,B 0,C 180,E1 -9688.772,E2 -9688.772} C_VEL
LIN {X 0,Y 429.904,Z 647.291,A -85,B 0,C 180,E1 -9689.551,E2 -9689.551} C_VEL
LIN {X 0,Y 429.338,Z 659.132,A -85,B 0,C 180,E1 -9690.451,E2 -9690.451} C_VEL
LIN {X 0,Y 428.63,Z 671.415,A -85,B 0,C 180,E1 -9691.609,E2 -9691.609} C_VEL
LIN {X 0,Y 427.907,Z 682.477,A -85,B 0,C 180,E1 -9692.886,E2 -9692.886} C_VEL
LIN {X 0,Y 427.336,Z 691.608,A -85,B 0,C 180,E1 -9694.163,E2 -9694.163} C_VEL
LIN {X 0,Y 426.705,Z 700.659,A -85,B 0,C 180,E1 -9695.685,E2 -9695.685} C_VEL
LIN {X 0,Y 426.25,Z 707.734,A -85,B 0,C 180,E1 -9697.139,E2 -9697.139} C_VEL
LIN {X 0,Y 425.805,Z 714.005,A -85,B 0,C 180,E1 -9698.709,E2 -9698.709} C_VEL
LIN {X 0,Y 425.542,Z 719.012,A -85,B 0,C 180,E1 -9700.282,E2 -9700.282} C_VEL
LIN {X 0,Y 425.315,Z 722.547,A -85,B 0,C 180,E1 -9701.702,E2 -9701.702} C_VEL
LIN {X 0,Y 425.096,Z 726.139,A -85,B 0,C 180,E1 -9703.677,E2 -9703.677} C_VEL
LIN {X 0,Y 425.03,Z 728.14,A -85,B 0,C 180,E1 -9705.64,E2 -9705.64} C_VEL
LIN {X 0,Y 425.103,Z 728.699,A -85,B 0,C 180,E1 -9707.589,E2 -9707.589} C_VEL
LIN {X 0,Y 425.158,Z 727.871,A -85,B 0,C 180,E1 -9709.524,E2 -9709.524} C_VEL
LIN {X 0,Y 425.374,Z 725.62,A -85,B 0,C 180,E1 -9711.449,E2 -9711.449} C_VEL
LIN {X 0,Y 425.749,Z 721.842,A -85,B 0,C 180,E1 -9713.365,E2 -9713.365} C_VEL
LIN {X 0,Y 426.111,Z 716.539,A -85,B 0,C 180,E1 -9715.27,E2 -9715.27} C_VEL
LIN {X 0,Y 426.538,Z 711.407,A -85,B 0,C 180,E1 -9716.694,E2 -9716.694} C_VEL
LIN {X 0,Y 427.14,Z 704.025,A -85,B 0,C 180,E1 -9718.35,E2 -9718.35} C_VEL
LIN {X 0,Y 427.772,Z 696.243,A -85,B 0,C 180,E1 -9719.765,E2 -9719.765} C_VEL
LIN {X 0,Y 428.535,Z 686.806,A -85,B 0,C 180,E1 -9721.175,E2 -9721.175} C_VEL
LIN {X 0,Y 429.196,Z 676.298,A -85,B 0,C 180,E1 -9722.458,E2 -9722.458} C_VEL
LIN {X 0,Y 429.981,Z 664.387,A -85,B 0,C 180,E1 -9723.632,E2 -9723.632} C_VEL
LIN {X 0,Y 430.643,Z 652.613,A -85,B 0,C 180,E1 -9724.564,E2 -9724.564} C_VEL
LIN {X 0,Y 431.042,Z 640.668,A -85,B 0,C 180,E1 -9725.321,E2 -9725.321} C_VEL
LIN {X 0,Y 431.387,Z 626.756,A -85,B 0,C 180,E1 -9725.991,E2 -9725.991} C_VEL
LIN {X 0,Y 431.525,Z 612.616,A -85,B 0,C 180,E1 -9726.459,E2 -9726.459} C_VEL
LIN {X 0,Y 431.646,Z 587.229,A -85,B 0,C 180,E1 -9726.957,E2 -9726.957} C_VEL
LIN {X 0,Y 431.861,Z 563.374,A -85,B 0,C 180,E1 -9727.392,E2 -9727.392} C_VEL
LIN {X 0,Y 426.159,Z 549.709,A -85,B 0,C 180,E1 -9727.981,E2 -9727.981} C_VEL
LIN {X 0,Y 425.505,Z 547.485,A -85,B 0,C 180,E1 -9728.086,E2 -9728.086} C_VEL
LIN {X 0,Y 425.365,Z 547.503,A -85,B 0,C 180,E1 -9731.436,E2 -9731.436} C_VEL
LIN {X 0,Y 425.35,Z 547.504,A -85,B 0,C 180,E1 -9734.35,E2 -9734.35} C_VEL
LIN {X 0,Y 425.339,Z 547.508,A -85,B 0,C 180,E1 -9737.303,E2 -9737.303} C_VEL
LIN {X 0,Y 425.293,Z 547.508,A -85,B 0,C 180,E1 -9740.306,E2 -9740.306} C_VEL
LIN {X 0,Y 425.304,Z 547.507,A -85,B 0,C 180,E1 -9743.366,E2 -9743.366} C_VEL
LIN {X 0,Y 425.346,Z 547.499,A -85,B 0,C 180,E1 -9746.845,E2 -9746.845} C_VEL
LIN {X 0,Y 425.316,Z 547.5,A -85,B 0,C 180,E1 -9749.718,E2 -9749.718} C_VEL
LIN {X 0,Y 425.28,Z 547.504,A -85,B 0,C 180,E1 -9753.049,E2 -9753.049} C_VEL
LIN {X 0,Y 425.282,Z 547.505,A -85,B 0,C 180,E1 -9755.93,E2 -9755.93} C_VEL
LIN {X 0,Y 425.302,Z 547.506,A -85,B 0,C 180,E1 -9759.045,E2 -9759.045} C_VEL
LIN {X 0,Y 425.277,Z 547.507,A -85,B 0,C 180,E1 -9762.653,E2 -9762.653} C_VEL
LIN {X 0,Y 425.26,Z 547.509,A -85,B 0,C 180,E1 -9766.045,E2 -9766.045} C_VEL
LIN {X 0,Y 425.273,Z 547.506,A -85,B 0,C 180,E1 -9768.622,E2 -9768.622} C_VEL
LIN {X 0,Y 425.313,Z 547.51,A -85,B 0,C 180,E1 -9771.104,E2 -9771.104} C_VEL
LIN {X 0,Y 425.347,Z 547.708,A -85,B 0,C 180,E1 -9773.78,E2 -9773.78} C_VEL
LIN {X 0,Y 428.789,Z 563.48,A -85,B 0,C 180,E1 -9777.257,E2 -9777.257} C_VEL
LIN {X 0,Y 429.747,Z 569.113,A -85,B 0,C 180,E1 -9778.445,E2 -9778.445} C_VEL
LIN {X 0,Y 428.41,Z 587.622,A -85,B 0,C 180,E1 -9782.052,E2 -9782.052} C_VEL
LIN {X 0,Y 427.205,Z 606.764,A -85,B 0,C 180,E1 -9785.716,E2 -9785.716} C_VEL
LIN {X 0,Y 426.354,Z 624.168,A -85,B 0,C 180,E1 -9788.991,E2 -9788.991} C_VEL
LIN {X 0,Y 425.984,Z 632.793,A -85,B 0,C 180,E1 -9790.598,E2 -9790.598} C_VEL
LIN {X 0,Y 430.916,Z 672.807,A -85,B 0,C 180,E1 -9791.705,E2 -9791.705} C_VEL
LIN {X 0,Y 429.336,Z 746.703,A -85,B 0,C 180,E1 -9793.293,E2 -9793.293} C_VEL
LIN {X 0,Y 428.759,Z 760.05,A -85,B 0,C 180,E1 -9793.76,E2 -9793.76} C_VEL
LIN {X 0,Y 427.981,Z 773.034,A -85,B 0,C 180,E1 -9794.402,E2 -9794.402} C_VEL
LIN {X 0,Y 427.138,Z 785.442,A -85,B 0,C 180,E1 -9795.225,E2 -9795.225} C_VEL
LIN {X 0,Y 426.478,Z 796.749,A -85,B 0,C 180,E1 -9796.177,E2 -9796.177} C_VEL
LIN {X 0,Y 426.006,Z 806.333,A -85,B 0,C 180,E1 -9797.164,E2 -9797.164} C_VEL
LIN {X 0,Y 425.423,Z 815.685,A -85,B 0,C 180,E1 -9798.325,E2 -9798.325} C_VEL
LIN {X 0,Y 424.9,Z 825.033,A -85,B 0,C 180,E1 -9799.758,E2 -9799.758} C_VEL
LIN {X 0,Y 424.687,Z 832.621,A -85,B 0,C 180,E1 -9801.195,E2 -9801.195} C_VEL
LIN {X 0,Y 424.589,Z 837.778,A -85,B 0,C 180,E1 -9802.391,E2 -9802.391} C_VEL
LIN {X 0,Y 424.579,Z 842.211,A -85,B 0,C 180,E1 -9803.641,E2 -9803.641} C_VEL
LIN {X 0,Y 424.64,Z 846.589,A -85,B 0,C 180,E1 -9805.254,E2 -9805.254} C_VEL
LIN {X 0,Y 424.687,Z 848.535,A -85,B 0,C 180,E1 -9806.205,E2 -9806.205} C_VEL
LIN {X 0,Y 424.652,Z 850.006,A -85,B 0,C 180,E1 -9807.155,E2 -9807.155} C_VEL
LIN {X 0,Y 424.662,Z 850.994,A -85,B 0,C 180,E1 -9808.104,E2 -9808.104} C_VEL
LIN {X 0,Y 424.675,Z 851.555,A -85,B 0,C 180,E1 -9809.052,E2 -9809.052} C_VEL
LIN {X 0,Y 424.895,Z 851.718,A -85,B 0,C 180,E1 -9810.001,E2 -9810.001} C_VEL
LIN {X 0,Y 424.697,Z 851.382,A -85,B 0,C 180,E1 -9810.949,E2 -9810.949} C_VEL
LIN {X 0,Y 424.708,Z 850.603,A -85,B 0,C 180,E1 -9811.897,E2 -9811.897} C_VEL
LIN {X 0,Y 424.714,Z 849.39,A -85,B 0,C 180,E1 -9812.846,E2 -9812.846} C_VEL
LIN {X 0,Y 424.771,Z 846.728,A -85,B 0,C 180,E1 -9814.27,E2 -9814.27} C_VEL
LIN {X 0,Y 424.648,Z 842.959,A -85,B 0,C 180,E1 -9815.699,E2 -9815.699} C_VEL
LIN {X 0,Y 424.665,Z 837.197,A -85,B 0,C 180,E1 -9817.346,E2 -9817.346} C_VEL
LIN {X 0,Y 424.733,Z 830.657,A -85,B 0,C 180,E1 -9818.805,E2 -9818.805} C_VEL
LIN {X 0,Y 424.917,Z 822.67,A -85,B 0,C 180,E1 -9820.242,E2 -9820.242} C_VEL
LIN {X 0,Y 425.334,Z 812.833,A -85,B 0,C 180,E1 -9821.679,E2 -9821.679} C_VEL
LIN {X 0,Y 425.718,Z 804.104,A -85,B 0,C 180,E1 -9822.734,E2 -9822.734} C_VEL
LIN {X 0,Y 426.493,Z 791.944,A -85,B 0,C 180,E1 -9823.946,E2 -9823.946} C_VEL
LIN {X 0,Y 427.041,Z 781.698,A -85,B 0,C 180,E1 -9824.779,E2 -9824.779} C_VEL
LIN {X 0,Y 427.974,Z 768.024,A -85,B 0,C 180,E1 -9825.661,E2 -9825.661} C_VEL
LIN {X 0,Y 428.737,Z 754.993,A -85,B 0,C 180,E1 -9826.304,E2 -9826.304} C_VEL
LIN {X 0,Y 429.355,Z 741.028,A -85,B 0,C 180,E1 -9826.799,E2 -9826.799} C_VEL
LIN {X 0,Y 429.875,Z 718.811,A -85,B 0,C 180,E1 -9827.291,E2 -9827.291} C_VEL
LIN {X 0,Y 430.71,Z 671.297,A -85,B 0,C 180,E1 -9828.277,E2 -9828.277} C_VEL
LIN {X 0,Y 429.337,Z 654.014,A -85,B 0,C 180,E1 -9828.739,E2 -9828.739} C_VEL
LIN {X 0,Y 427.727,Z 633.271,A -85,B 0,C 180,E1 -9829.31,E2 -9829.31} C_VEL
LIN {X 0,Y 425.601,Z 615.489,A -85,B 0,C 180,E1 -9829.884,E2 -9829.884} C_VEL
LIN {X 0,Y 425.833,Z 597.029,A -85,B 0,C 180,E1 -9833.082,E2 -9833.082} C_VEL
LIN {X 0,Y 426.203,Z 578.075,A -85,B 0,C 180,E1 -9836.438,E2 -9836.438} C_VEL
LIN {X 0,Y 426.684,Z 560.663,A -85,B 0,C 180,E1 -9839.613,E2 -9839.613} C_VEL
LIN {X 0,Y 426.639,Z 554.846,A -85,B 0,C 180,E1 -9840.708,E2 -9840.708} C_VEL
LIN {X 0,Y 425.378,Z 547.502,A -85,B 0,C 180,E1 -9842.199,E2 -9842.199} C_VEL
LIN {X 0,Y 425.304,Z 547.508,A -85,B 0,C 180,E1 -9845.336,E2 -9845.336} C_VEL
LIN {X 0,Y 425.298,Z 547.51,A -85,B 0,C 180,E1 -9849.043,E2 -9849.043} C_VEL
LIN {X 0,Y 425.279,Z 547.51,A -85,B 0,C 180,E1 -9852.653,E2 -9852.653} C_VEL
LIN {X 0,Y 425.266,Z 547.511,A -85,B 0,C 180,E1 -9856.044,E2 -9856.044} C_VEL
LIN {X 0,Y 425.279,Z 547.51,A -85,B 0,C 180,E1 -9858.621,E2 -9858.621} C_VEL
LIN {X 0,Y 425.314,Z 547.507,A -85,B 0,C 180,E1 -9861.103,E2 -9861.103} C_VEL
LIN {X 0,Y 425.304,Z 547.508,A -85,B 0,C 180,E1 -9864.664,E2 -9864.664} C_VEL
LIN {X 0,Y 425.27,Z 547.511,A -85,B 0,C 180,E1 -9868.073,E2 -9868.073} C_VEL
LIN {X 0,Y 425.336,Z 547.503,A -85,B 0,C 180,E1 -9871.368,E2 -9871.368} C_VEL
LIN {X 0,Y 425.3,Z 547.512,A -85,B 0,C 180,E1 -9874.555,E2 -9874.555} C_VEL
LIN {X 0,Y 425.292,Z 547.512,A -85,B 0,C 180,E1 -9877.661,E2 -9877.661} C_VEL
LIN {X 0,Y 425.33,Z 547.505,A -85,B 0,C 180,E1 -9879.525,E2 -9879.525} C_VEL
LIN {X 0,Y 426.364,Z 550.447,A -85,B 0,C 180,E1 -9879.667,E2 -9879.667} C_VEL
LIN {X 0,Y 432.501,Z 564.189,A -85,B 0,C 180,E1 -9880.308,E2 -9880.308} C_VEL
LIN {X 0,Y 432.983,Z 566.193,A -85,B 0,C 180,E1 -9880.372,E2 -9880.372} C_VEL
LIN {X 0,Y 432.891,Z 598.133,A -85,B 0,C 180,E1 -9880.959,E2 -9880.959} C_VEL
LIN {X 0,Y 432.867,Z 613.143,A -85,B 0,C 180,E1 -9881.425,E2 -9881.425} C_VEL
LIN {X 0,Y 432.624,Z 627.793,A -85,B 0,C 180,E1 -9882.082,E2 -9882.082} C_VEL
LIN {X 0,Y 432.177,Z 640.946,A -85,B 0,C 180,E1 -9882.857,E2 -9882.857} C_VEL
LIN {X 0,Y 431.573,Z 653.745,A -85,B 0,C 180,E1 -9883.807,E2 -9883.807} C_VEL
LIN {X 0,Y 430.89,Z 665.529,A -85,B 0,C 180,E1 -9884.872,E2 -9884.872} C_VEL
LIN {X 0,Y 430.135,Z 676.367,A -85,B 0,C 180,E1 -9886.054,E2 -9886.054} C_VEL
LIN {X 0,Y 429.24,Z 687.141,A -85,B 0,C 180,E1 -9887.47,E2 -9887.47} C_VEL
LIN {X 0,Y 428.474,Z 696.101,A -85,B 0,C 180,E1 -9888.888,E2 -9888.888} C_VEL
LIN {X 0,Y 427.708,Z 704.752,A -85,B 0,C 180,E1 -9890.542,E2 -9890.542} C_VEL
LIN {X 0,Y 426.897,Z 712.749,A -85,B 0,C 180,E1 -9892.432,E2 -9892.432} C_VEL
LIN {X 0,Y 426.531,Z 717.604,A -85,B 0,C 180,E1 -9893.851,E2 -9893.851} C_VEL
LIN {X 0,Y 426.09,Z 722.768,A -85,B 0,C 180,E1 -9895.743,E2 -9895.743} C_VEL
LIN {X 0,Y 425.704,Z 725.748,A -85,B 0,C 180,E1 -9897.161,E2 -9897.161} C_VEL
LIN {X 0,Y 425.436,Z 728.576,A -85,B 0,C 180,E1 -9899.053,E2 -9899.053} C_VEL
LIN {X 0,Y 425.298,Z 730.182,A -85,B 0,C 180,E1 -9900.946,E2 -9900.946} C_VEL
LIN {X 0,Y 425.29,Z 730.582,A -85,B 0,C 180,E1 -9902.841,E2 -9902.841} C_VEL
LIN {X 0,Y 425.179,Z 729.804,A -85,B 0,C 180,E1 -9904.74,E2 -9904.74} C_VEL
LIN {X 0,Y 425.361,Z 727.804,A -85,B 0,C 180,E1 -9906.641,E2 -9906.641} C_VEL
LIN {X 0,Y 425.474,Z 724.587,A -85,B 0,C 180,E1 -9908.549,E2 -9908.549} C_VEL
LIN {X 0,Y 425.704,Z 720.051,A -85,B 0,C 180,E1 -9910.463,E2 -9910.463} C_VEL
LIN {X 0,Y 426.078,Z 714.07,A -85,B 0,C 180,E1 -9912.382,E2 -9912.382} C_VEL
LIN {X 0,Y 426.534,Z 707.584,A -85,B 0,C 180,E1 -9914.041,E2 -9914.041} C_VEL
LIN {X 0,Y 427.151,Z 699.447,A -85,B 0,C 180,E1 -9915.752,E2 -9915.752} C_VEL
LIN {X 0,Y 427.836,Z 690.131,A -85,B 0,C 180,E1 -9917.373,E2 -9917.373} C_VEL
LIN {X 0,Y 428.534,Z 679.605,A -85,B 0,C 180,E1 -9918.899,E2 -9918.899} C_VEL
LIN {X 0,Y 429.262,Z 668.56,A -85,B 0,C 180,E1 -9920.234,E2 -9920.234} C_VEL
LIN {X 0,Y 430.041,Z 656.551,A -85,B 0,C 180,E1 -9921.446,E2 -9921.446} C_VEL
LIN {X 0,Y 430.802,Z 643.369,A -85,B 0,C 180,E1 -9922.542,E2 -9922.542} C_VEL
LIN {X 0,Y 431.39,Z 629.758,A -85,B 0,C 180,E1 -9923.46,E2 -9923.46} C_VEL
LIN {X 0,Y 431.972,Z 615.022,A -85,B 0,C 180,E1 -9924.236,E2 -9924.236} C_VEL
LIN {X 0,Y 432.25,Z 600.291,A -85,B 0,C 180,E1 -9924.818,E2 -9924.818} C_VEL
LIN {X 0,Y 432.37,Z 585.42,A -85,B 0,C 180,E1 -9925.219,E2 -9925.219} C_VEL
LIN {X 0,Y 432.439,Z 566.583,A -85,B 0,C 180,E1 -9925.588,E2 -9925.588} C_VEL
LIN {X 0,Y 425.473,Z 548.106,A -85,B 0,C 180,E1 -9926.252,E2 -9926.252} C_VEL
LIN {X 0,Y 425.349,Z 547.503,A -85,B 0,C 180,E1 -9926.293,E2 -9926.293} C_VEL
LIN {X 0,Y 425.292,Z 547.51,A -85,B 0,C 180,E1 -9929.719,E2 -9929.719} C_VEL
LIN {X 0,Y 425.283,Z 547.505,A -85,B 0,C 180,E1 -9933.047,E2 -9933.047} C_VEL
LIN {X 0,Y 425.283,Z 547.51,A -85,B 0,C 180,E1 -9935.928,E2 -9935.928} C_VEL
LIN {X 0,Y 425.294,Z 547.504,A -85,B 0,C 180,E1 -9939.042,E2 -9939.042} C_VEL
LIN {X 0,Y 425.275,Z 547.509,A -85,B 0,C 180,E1 -9942.652,E2 -9942.652} C_VEL
LIN {X 0,Y 425.262,Z 547.512,A -85,B 0,C 180,E1 -9946.044,E2 -9946.044} C_VEL
LIN {X 0,Y 425.275,Z 547.511,A -85,B 0,C 180,E1 -9948.621,E2 -9948.621} C_VEL
LIN {X 0,Y 425.315,Z 547.502,A -85,B 0,C 180,E1 -9951.103,E2 -9951.103} C_VEL
LIN {X 0,Y 425.299,Z 547.509,A -85,B 0,C 180,E1 -9954.664,E2 -9954.664} C_VEL
LIN {X 0,Y 425.264,Z 547.51,A -85,B 0,C 180,E1 -9958.072,E2 -9958.072} C_VEL
LIN {X 0,Y 425.331,Z 547.5,A -85,B 0,C 180,E1 -9961.367,E2 -9961.367} C_VEL
LIN {X 0,Y 425.295,Z 547.51,A -85,B 0,C 180,E1 -9964.554,E2 -9964.554} C_VEL
LIN {X 0,Y 425.287,Z 547.505,A -85,B 0,C 180,E1 -9967.661,E2 -9967.661} C_VEL
LIN {X 0,Y 425.361,Z 547.502,A -85,B 0,C 180,E1 -9970.703,E2 -9970.703} C_VEL
LIN {X 0,Y 425.387,Z 547.492,A -85,B 0,C 180,E1 -9973.688,E2 -9973.688} C_VEL
LIN {X 0,Y 425.411,Z 547.49,A -85,B 0,C 180,E1 -9977.598,E2 -9977.598} C_VEL
LIN {X 0,Y 425.441,Z 547.488,A -85,B 0,C 180,E1 -9981.449,E2 -9981.449} C_VEL
LIN {X 0,Y 425.553,Z 547.472,A -85,B 0,C 180,E1 -9984.313,E2 -9984.313} C_VEL
LIN {X 0,Y 425.573,Z 547.469,A -85,B 0,C 180,E1 -9988.107,E2 -9988.107} C_VEL
LIN {X 0,Y 425.642,Z 547.461,A -85,B 0,C 180,E1 -9989.722,E2 -9989.722} C_VEL
LIN {X 0,Y 425.396,Z 547.492,A -85,B 0,C 180,E1 -9990.251,E2 -9990.251} C_VEL
LIN {X 0,Y 424.044,Z 547.666,A -85,B 0,C 180,E1 -9991.029,E2 -9991.029} C_VEL
LIN {X 0,Y 419.494,Z 548.23,A -85,B 0,C 180,E1 -9992.824,E2 -9992.824} C_VEL
LIN {X 0,Y 418.377,Z 548.369,A -85,B 0,C 180,E1 -9993.626,E2 -9993.626} C_VEL
LIN {X 0,Y 418.288,Z 548.377,A -85,B 0,C 180,E1 -9993.898,E2 -9993.898} C_VEL
LIN {X 0,Y 418.507,Z 548.351,A -85,B 0,C 180,E1 -9995.782,E2 -9995.782} C_VEL
LIN {X 0,Y 418.398,Z 548.364,A -85,B 0,C 180,E1 -9998.695,E2 -9998.695} C_VEL
LIN {X 0,Y 418.332,Z 548.375,A -85,B 0,C 180,E1 -10001.63,E2 -10001.63} C_VEL
LIN {X 0,Y 418.304,Z 548.375,A -85,B 0,C 180,E1 -10004.596,E2 -10004.596} C_VEL
LIN {X 0,Y 418.285,Z 548.383,A -85,B 0,C 180,E1 -10007.603,E2 -10007.603} C_VEL
LIN {X 0,Y 418.246,Z 548.382,A -85,B 0,C 180,E1 -10010.662,E2 -10010.662} C_VEL
LIN {X 0,Y 418.284,Z 548.382,A -85,B 0,C 180,E1 -10013.781,E2 -10013.781} C_VEL
LIN {X 0,Y 418.305,Z 548.376,A -85,B 0,C 180,E1 -10017.07,E2 -10017.07} C_VEL
LIN {X 0,Y 418.258,Z 548.382,A -85,B 0,C 180,E1 -10020.27,E2 -10020.27} C_VEL
LIN {X 0,Y 418.245,Z 548.389,A -85,B 0,C 180,E1 -10023.677,E2 -10023.677} C_VEL
LIN {X 0,Y 418.242,Z 548.384,A -85,B 0,C 180,E1 -10027.223,E2 -10027.223} C_VEL
LIN {X 0,Y 418.259,Z 548.385,A -85,B 0,C 180,E1 -10029.68,E2 -10029.68} C_VEL
LIN {X 0,Y 418.24,Z 548.385,A -85,B 0,C 180,E1 -10032.323,E2 -10032.323} C_VEL
LIN {X 0,Y 418.254,Z 548.381,A -85,B 0,C 180,E1 -10035.112,E2 -10035.112} C_VEL
LIN {X 0,Y 418.287,Z 548.381,A -85,B 0,C 180,E1 -10037.773,E2 -10037.773} C_VEL
LIN {X 0,Y 418.262,Z 548.381,A -85,B 0,C 180,E1 -10041.56,E2 -10041.56} C_VEL
LIN {X 0,Y 418.254,Z 548.381,A -85,B 0,C 180,E1 -10045.159,E2 -10045.159} C_VEL
LIN {X 0,Y 418.29,Z 548.38,A -85,B 0,C 180,E1 -10046.022,E2 -10046.022} C_VEL
LIN {X 0,Y 424.599,Z 565.552,A -85,B 0,C 180,E1 -10046.646,E2 -10046.646} C_VEL
LIN {X 0,Y 424.144,Z 607.417,A -85,B 0,C 180,E1 -10047.456,E2 -10047.456} C_VEL
LIN {X 0,Y 423.965,Z 620.694,A -85,B 0,C 180,E1 -10047.875,E2 -10047.875} C_VEL
LIN {X 0,Y 423.603,Z 634.39,A -85,B 0,C 180,E1 -10048.493,E2 -10048.493} C_VEL
LIN {X 0,Y 423.119,Z 647.16,A -85,B 0,C 180,E1 -10049.256,E2 -10049.256} C_VEL
LIN {X 0,Y 422.511,Z 659.642,A -85,B 0,C 180,E1 -10050.203,E2 -10050.203} C_VEL
LIN {X 0,Y 421.773,Z 671.999,A -85,B 0,C 180,E1 -10051.377,E2 -10051.377} C_VEL
LIN {X 0,Y 421.011,Z 683.14,A -85,B 0,C 180,E1 -10052.674,E2 -10052.674} C_VEL
LIN {X 0,Y 420.419,Z 692.34,A -85,B 0,C 180,E1 -10053.972,E2 -10053.972} C_VEL
LIN {X 0,Y 419.755,Z 701.451,A -85,B 0,C 180,E1 -10055.52,E2 -10055.52} C_VEL
LIN {X 0,Y 419.207,Z 709.565,A -85,B 0,C 180,E1 -10057.229,E2 -10057.229} C_VEL
LIN {X 0,Y 418.772,Z 715.756,A -85,B 0,C 180,E1 -10058.85,E2 -10058.85} C_VEL
LIN {X 0,Y 418.511,Z 720.433,A -85,B 0,C 180,E1 -10060.376,E2 -10060.376} C_VEL
LIN {X 0,Y 418.257,Z 724.071,A -85,B 0,C 180,E1 -10061.89,E2 -10061.89} C_VEL
LIN {X 0,Y 418.092,Z 726.741,A -85,B 0,C 180,E1 -10063.396,E2 -10063.396} C_VEL
LIN {X 0,Y 418.014,Z 729.006,A -85,B 0,C 180,E1 -10065.393,E2 -10065.393} C_VEL
LIN {X 0,Y 418.086,Z 729.75,A -85,B 0,C 180,E1 -10067.378,E2 -10067.378} C_VEL
LIN {X 0,Y 418.132,Z 729.091,A -85,B 0,C 180,E1 -10069.346,E2 -10069.346} C_VEL
LIN {X 0,Y 418.355,Z 727.021,A -85,B 0,C 180,E1 -10071.304,E2 -10071.304} C_VEL
LIN {X 0,Y 418.74,Z 723.493,A -85,B 0,C 180,E1 -10073.253,E2 -10073.253} C_VEL
LIN {X 0,Y 419.129,Z 718.381,A -85,B 0,C 180,E1 -10075.191,E2 -10075.191} C_VEL
LIN {X 0,Y 419.582,Z 713.437,A -85,B 0,C 180,E1 -10076.64,E2 -10076.64} C_VEL
LIN {X 0,Y 420.209,Z 706.251,A -85,B 0,C 180,E1 -10078.323,E2 -10078.323} C_VEL
LIN {X 0,Y 420.851,Z 698.69,A -85,B 0,C 180,E1 -10079.761,E2 -10079.761} C_VEL
LIN {X 0,Y 421.706,Z 689.12,A -85,B 0,C 180,E1 -10081.248,E2 -10081.248} C_VEL
LIN {X 0,Y 422.315,Z 679.34,A -85,B 0,C 180,E1 -10082.504,E2 -10082.504} C_VEL
LIN {X 0,Y 423.152,Z 667.967,A -85,B 0,C 180,E1 -10083.69,E2 -10083.69} C_VEL
LIN {X 0,Y 423.879,Z 656.276,A -85,B 0,C 180,E1 -10084.674,E2 -10084.674} C_VEL
LIN {X 0,Y 424.378,Z 643.088,A -85,B 0,C 180,E1 -10085.556,E2 -10085.556} C_VEL
LIN {X 0,Y 424.779,Z 629.338,A -85,B 0,C 180,E1 -10086.249,E2 -10086.249} C_VEL
LIN {X 0,Y 424.917,Z 615.123,A -85,B 0,C 180,E1 -10086.748,E2 -10086.748} C_VEL
LIN {X 0,Y 424.928,Z 594.277,A -85,B 0,C 180,E1 -10087.184,E2 -10087.184} C_VEL
LIN {X 0,Y 425.251,Z 564.942,A -85,B 0,C 180,E1 -10087.729,E2 -10087.729} C_VEL
LIN {X 0,Y 419.449,Z 551.271,A -85,B 0,C 180,E1 -10088.354,E2 -10088.354} C_VEL
LIN {X 0,Y 418.398,Z 548.369,A -85,B 0,C 180,E1 -10088.508,E2 -10088.508} C_VEL
LIN {X 0,Y 418.328,Z 548.38,A -85,B 0,C 180,E1 -10091.631,E2 -10091.631} C_VEL
LIN {X 0,Y 418.303,Z 548.382,A -85,B 0,C 180,E1 -10094.597,E2 -10094.597} C_VEL
LIN {X 0,Y 418.285,Z 548.385,A -85,B 0,C 180,E1 -10097.604,E2 -10097.604} C_VEL
LIN {X 0,Y 418.247,Z 548.386,A -85,B 0,C 180,E1 -10100.664,E2 -10100.664} C_VEL
LIN {X 0,Y 418.285,Z 548.382,A -85,B 0,C 180,E1 -10103.782,E2 -10103.782} C_VEL
LIN {X 0,Y 418.307,Z 548.378,A -85,B 0,C 180,E1 -10107.071,E2 -10107.071} C_VEL
LIN {X 0,Y 418.259,Z 548.377,A -85,B 0,C 180,E1 -10110.271,E2 -10110.271} C_VEL
LIN {X 0,Y 418.246,Z 548.381,A -85,B 0,C 180,E1 -10113.678,E2 -10113.678} C_VEL
LIN {X 0,Y 418.243,Z 548.383,A -85,B 0,C 180,E1 -10117.224,E2 -10117.224} C_VEL
LIN {X 0,Y 418.254,Z 548.383,A -85,B 0,C 180,E1 -10119.682,E2 -10119.682} C_VEL
LIN {X 0,Y 418.231,Z 548.384,A -85,B 0,C 180,E1 -10122.322,E2 -10122.322} C_VEL
LIN {X 0,Y 418.237,Z 548.39,A -85,B 0,C 180,E1 -10125.11,E2 -10125.11} C_VEL
LIN {X 0,Y 418.239,Z 548.384,A -85,B 0,C 180,E1 -10127.768,E2 -10127.768} C_VEL
LIN {X 0,Y 418.257,Z 548.385,A -85,B 0,C 180,E1 -10130.619,E2 -10130.619} C_VEL
LIN {X 0,Y 418.288,Z 548.533,A -85,B 0,C 180,E1 -10133.511,E2 -10133.511} C_VEL
LIN {X 0,Y 421.536,Z 563.638,A -85,B 0,C 180,E1 -10136.906,E2 -10136.906} C_VEL
LIN {X 0,Y 422.606,Z 568.728,A -85,B 0,C 180,E1 -10138.01,E2 -10138.01} C_VEL
LIN {X 0,Y 422.654,Z 572.054,A -85,B 0,C 180,E1 -10138.693,E2 -10138.693} C_VEL
LIN {X 0,Y 421.348,Z 589.534,A -85,B 0,C 180,E1 -10142.159,E2 -10142.159} C_VEL
LIN {X 0,Y 420.138,Z 608.287,A -85,B 0,C 180,E1 -10145.806,E2 -10145.806} C_VEL
LIN {X 0,Y 419.23,Z 625.642,A -85,B 0,C 180,E1 -10149.131,E2 -10149.131} C_VEL
LIN {X 0,Y 418.975,Z 631.696,A -85,B 0,C 180,E1 -10150.257,E2 -10150.257} C_VEL
LIN {X 0,Y 424.112,Z 673.123,A -85,B 0,C 180,E1 -10151.438,E2 -10151.438} C_VEL
LIN {X 0,Y 422.463,Z 745.786,A -85,B 0,C 180,E1 -10153.044,E2 -10153.044} C_VEL
LIN {X 0,Y 421.934,Z 758.323,A -85,B 0,C 180,E1 -10153.489,E2 -10153.489} C_VEL
LIN {X 0,Y 421.118,Z 771.447,A -85,B 0,C 180,E1 -10154.141,E2 -10154.141} C_VEL
LIN {X 0,Y 420.269,Z 783.985,A -85,B 0,C 180,E1 -10154.978,E2 -10154.978} C_VEL
LIN {X 0,Y 419.442,Z 796.635,A -85,B 0,C 180,E1 -10156.063,E2 -10156.063} C_VEL
LIN {X 0,Y 418.892,Z 807.237,A -85,B 0,C 180,E1 -10157.207,E2 -10157.207} C_VEL
LIN {X 0,Y 418.328,Z 816.107,A -85,B 0,C 180,E1 -10158.37,E2 -10158.37} C_VEL
LIN {X 0,Y 417.811,Z 825.215,A -85,B 0,C 180,E1 -10159.828,E2 -10159.828} C_VEL
LIN {X 0,Y 417.612,Z 832.599,A -85,B 0,C 180,E1 -10161.289,E2 -10161.289} C_VEL
LIN {X 0,Y 417.483,Z 838.479,A -85,B 0,C 180,E1 -10162.747,E2 -10162.747} C_VEL
LIN {X 0,Y 417.495,Z 843.097,A -85,B 0,C 180,E1 -10164.204,E2 -10164.204} C_VEL
LIN {X 0,Y 417.592,Z 845.524,A -85,B 0,C 180,E1 -10165.173,E2 -10165.173} C_VEL
LIN {X 0,Y 417.65,Z 847.483,A -85,B 0,C 180,E1 -10166.141,E2 -10166.141} C_VEL
LIN {X 0,Y 417.614,Z 848.972,A -85,B 0,C 180,E1 -10167.107,E2 -10167.107} C_VEL
LIN {X 0,Y 417.626,Z 849.973,A -85,B 0,C 180,E1 -10168.072,E2 -10168.072} C_VEL
LIN {X 0,Y 417.645,Z 850.537,A -85,B 0,C 180,E1 -10169.036,E2 -10169.036} C_VEL
LIN {X 0,Y 417.872,Z 850.703,A -85,B 0,C 180,E1 -10170.001,E2 -10170.001} C_VEL
LIN {X 0,Y 417.666,Z 850.371,A -85,B 0,C 180,E1 -10170.965,E2 -10170.965} C_VEL
LIN {X 0,Y 417.671,Z 849.592,A -85,B 0,C 180,E1 -10171.929,E2 -10171.929} C_VEL
LIN {X 0,Y 417.672,Z 848.376,A -85,B 0,C 180,E1 -10172.894,E2 -10172.894} C_VEL
LIN {X 0,Y 417.732,Z 845.712,A -85,B 0,C 180,E1 -10174.343,E2 -10174.343} C_VEL
LIN {X 0,Y 417.625,Z 840.854,A -85,B 0,C 180,E1 -10176.151,E2 -10176.151} C_VEL
LIN {X 0,Y 417.598,Z 835.092,A -85,B 0,C 180,E1 -10177.738,E2 -10177.738} C_VEL
LIN {X 0,Y 417.667,Z 828.381,A -85,B 0,C 180,E1 -10179.199,E2 -10179.199} C_VEL
LIN {X 0,Y 417.925,Z 820.106,A -85,B 0,C 180,E1 -10180.661,E2 -10180.661} C_VEL
LIN {X 0,Y 418.41,Z 809.973,A -85,B 0,C 180,E1 -10182.121,E2 -10182.121} C_VEL
LIN {X 0,Y 418.76,Z 801.286,A -85,B 0,C 180,E1 -10183.156,E2 -10183.156} C_VEL
LIN {X 0,Y 419.484,Z 790.995,A -85,B 0,C 180,E1 -10184.184,E2 -10184.184} C_VEL
LIN {X 0,Y 420.283,Z 779.219,A -85,B 0,C 180,E1 -10185.147,E2 -10185.147} C_VEL
LIN {X 0,Y 421.211,Z 765.318,A -85,B 0,C 180,E1 -10186.043,E2 -10186.043} C_VEL
LIN {X 0,Y 422.116,Z 751.955,A -85,B 0,C 180,E1 -10186.691,E2 -10186.691} C_VEL
LIN {X 0,Y 422.848,Z 736.325,A -85,B 0,C 180,E1 -10187.221,E2 -10187.221} C_VEL
LIN {X 0,Y 424.061,Z 671.67,A -85,B 0,C 180,E1 -10188.622,E2 -10188.622} C_VEL
LIN {X 0,Y 422.743,Z 653.866,A -85,B 0,C 180,E1 -10189.112,E2 -10189.112} C_VEL
LIN {X 0,Y 421.18,Z 633.361,A -85,B 0,C 180,E1 -10189.704,E2 -10189.704} C_VEL
LIN {X 0,Y 418.541,Z 612.725,A -85,B 0,C 180,E1 -10190.402,E2 -10190.402} C_VEL
LIN {X 0,Y 418.849,Z 593.861,A -85,B 0,C 180,E1 -10193.748,E2 -10193.748} C_VEL
LIN {X 0,Y 419.254,Z 574.201,A -85,B 0,C 180,E1 -10197.321,E2 -10197.321} C_VEL
LIN {X 0,Y 419.728,Z 559.116,A -85,B 0,C 180,E1 -10200.154,E2 -10200.154} C_VEL
LIN {X 0,Y 419.269,Z 553.273,A -85,B 0,C 180,E1 -10201.308,E2 -10201.308} C_VEL
LIN {X 0,Y 418.329,Z 548.381,A -85,B 0,C 180,E1 -10202.343,E2 -10202.343} C_VEL
LIN {X 0,Y 418.248,Z 548.385,A -85,B 0,C 180,E1 -10206.024,E2 -10206.024} C_VEL
LIN {X 0,Y 418.253,Z 548.383,A -85,B 0,C 180,E1 -10209.682,E2 -10209.682} C_VEL
LIN {X 0,Y 418.234,Z 548.386,A -85,B 0,C 180,E1 -10212.321,E2 -10212.321} C_VEL
LIN {X 0,Y 418.24,Z 548.389,A -85,B 0,C 180,E1 -10215.109,E2 -10215.109} C_VEL
LIN {X 0,Y 418.245,Z 548.385,A -85,B 0,C 180,E1 -10217.767,E2 -10217.767} C_VEL
LIN {X 0,Y 418.26,Z 548.384,A -85,B 0,C 180,E1 -10220.619,E2 -10220.619} C_VEL
LIN {X 0,Y 418.247,Z 548.386,A -85,B 0,C 180,E1 -10223.976,E2 -10223.976} C_VEL
LIN {X 0,Y 418.262,Z 548.385,A -85,B 0,C 180,E1 -10227.156,E2 -10227.156} C_VEL
LIN {X 0,Y 418.273,Z 548.385,A -85,B 0,C 180,E1 -10230.895,E2 -10230.895} C_VEL
LIN {X 0,Y 418.276,Z 548.387,A -85,B 0,C 180,E1 -10234.096,E2 -10234.096} C_VEL
LIN {X 0,Y 418.243,Z 548.39,A -85,B 0,C 180,E1 -10237.264,E2 -10237.264} C_VEL
LIN {X 0,Y 418.279,Z 548.384,A -85,B 0,C 180,E1 -10239.081,E2 -10239.081} C_VEL
LIN {X 0,Y 419.29,Z 551.279,A -85,B 0,C 180,E1 -10239.213,E2 -10239.213} C_VEL
LIN {X 0,Y 425.66,Z 564.959,A -85,B 0,C 180,E1 -10239.895,E2 -10239.895} C_VEL
LIN {X 0,Y 426.483,Z 567.517,A -85,B 0,C 180,E1 -10239.996,E2 -10239.996} C_VEL
LIN {X 0,Y 426.399,Z 599.1,A -85,B 0,C 180,E1 -10240.599,E2 -10240.599} C_VEL
LIN {X 0,Y 426.371,Z 614.389,A -85,B 0,C 180,E1 -10241.075,E2 -10241.075} C_VEL
LIN {X 0,Y 426.155,Z 628.01,A -85,B 0,C 180,E1 -10241.683,E2 -10241.683} C_VEL
LIN {X 0,Y 425.692,Z 641.368,A -85,B 0,C 180,E1 -10242.464,E2 -10242.464} C_VEL
LIN {X 0,Y 425.047,Z 654.664,A -85,B 0,C 180,E1 -10243.452,E2 -10243.452} C_VEL
LIN {X 0,Y 424.262,Z 667.378,A -85,B 0,C 180,E1 -10244.63,E2 -10244.63} C_VEL
LIN {X 0,Y 423.433,Z 678.088,A -85,B 0,C 180,E1 -10245.829,E2 -10245.829} C_VEL
LIN {X 0,Y 422.487,Z 688.779,A -85,B 0,C 180,E1 -10247.266,E2 -10247.266} C_VEL
LIN {X 0,Y 421.713,Z 697.696,A -85,B 0,C 180,E1 -10248.707,E2 -10248.707} C_VEL
LIN {X 0,Y 420.89,Z 706.288,A -85,B 0,C 180,E1 -10250.387,E2 -10250.387} C_VEL
LIN {X 0,Y 420.009,Z 714.201,A -85,B 0,C 180,E1 -10252.307,E2 -10252.307} C_VEL
LIN {X 0,Y 419.608,Z 719.001,A -85,B 0,C 180,E1 -10253.749,E2 -10253.749} C_VEL
LIN {X 0,Y 419.139,Z 724.084,A -85,B 0,C 180,E1 -10255.672,E2 -10255.672} C_VEL
LIN {X 0,Y 418.731,Z 727.007,A -85,B 0,C 180,E1 -10257.113,E2 -10257.113} C_VEL
LIN {X 0,Y 418.462,Z 729.769,A -85,B 0,C 180,E1 -10259.037,E2 -10259.037} C_VEL
LIN {X 0,Y 418.287,Z 731.308,A -85,B 0,C 180,E1 -10260.962,E2 -10260.962} C_VEL
LIN {X 0,Y 418.27,Z 731.641,A -85,B 0,C 180,E1 -10262.889,E2 -10262.889} C_VEL
LIN {X 0,Y 418.166,Z 730.795,A -85,B 0,C 180,E1 -10264.82,E2 -10264.82} C_VEL
LIN {X 0,Y 418.355,Z 728.705,A -85,B 0,C 180,E1 -10266.753,E2 -10266.753} C_VEL
LIN {X 0,Y 418.489,Z 725.387,A -85,B 0,C 180,E1 -10268.693,E2 -10268.693} C_VEL
LIN {X 0,Y 418.733,Z 720.739,A -85,B 0,C 180,E1 -10270.639,E2 -10270.639} C_VEL
LIN {X 0,Y 419.135,Z 714.631,A -85,B 0,C 180,E1 -10272.59,E2 -10272.59} C_VEL
LIN {X 0,Y 419.594,Z 708.012,A -85,B 0,C 180,E1 -10274.278,E2 -10274.278} C_VEL
LIN {X 0,Y 420.253,Z 699.717,A -85,B 0,C 180,E1 -10276.017,E2 -10276.017} C_VEL
LIN {X 0,Y 420.886,Z 691.295,A -85,B 0,C 180,E1 -10277.491,E2 -10277.491} C_VEL
LIN {X 0,Y 421.566,Z 681.3,A -85,B 0,C 180,E1 -10278.97,E2 -10278.97} C_VEL
LIN {X 0,Y 422.365,Z 670.368,A -85,B 0,C 180,E1 -10280.325,E2 -10280.325} C_VEL
LIN {X 0,Y 423.14,Z 658.604,A -85,B 0,C 180,E1 -10281.547,E2 -10281.547} C_VEL
LIN {X 0,Y 423.814,Z 647.097,A -85,B 0,C 180,E1 -10282.549,E2 -10282.549} C_VEL
LIN {X 0,Y 424.468,Z 633.144,A -85,B 0,C 180,E1 -10283.543,E2 -10283.543} C_VEL
LIN {X 0,Y 425.065,Z 618.696,A -85,B 0,C 180,E1 -10284.35,E2 -10284.35} C_VEL
LIN {X 0,Y 425.446,Z 603.256,A -85,B 0,C 180,E1 -10284.998,E2 -10284.998} C_VEL
LIN {X 0,Y 425.577,Z 588.527,A -85,B 0,C 180,E1 -10285.427,E2 -10285.427} C_VEL
LIN {X 0,Y 425.657,Z 568.238,A -85,B 0,C 180,E1 -10285.837,E2 -10285.837} C_VEL
LIN {X 0,Y 418.324,Z 548.376,A -85,B 0,C 180,E1 -10286.574,E2 -10286.574} C_VEL
LIN {X 0,Y 418.266,Z 548.382,A -85,B 0,C 180,E1 -10289.161,E2 -10289.161} C_VEL
LIN {X 0,Y 418.259,Z 548.381,A -85,B 0,C 180,E1 -10292.843,E2 -10292.843} C_VEL
LIN {X 0,Y 418.246,Z 548.389,A -85,B 0,C 180,E1 -10296.237,E2 -10296.237} C_VEL
LIN {X 0,Y 418.249,Z 548.383,A -85,B 0,C 180,E1 -10299.682,E2 -10299.682} C_VEL
LIN {X 0,Y 418.23,Z 548.391,A -85,B 0,C 180,E1 -10302.321,E2 -10302.321} C_VEL
LIN {X 0,Y 418.235,Z 548.383,A -85,B 0,C 180,E1 -10305.108,E2 -10305.108} C_VEL
LIN {X 0,Y 418.24,Z 548.384,A -85,B 0,C 180,E1 -10307.766,E2 -10307.766} C_VEL
LIN {X 0,Y 418.26,Z 548.385,A -85,B 0,C 180,E1 -10310.618,E2 -10310.618} C_VEL
LIN {X 0,Y 418.245,Z 548.384,A -85,B 0,C 180,E1 -10313.975,E2 -10313.975} C_VEL
LIN {X 0,Y 418.257,Z 548.382,A -85,B 0,C 180,E1 -10317.155,E2 -10317.155} C_VEL
LIN {X 0,Y 418.268,Z 548.383,A -85,B 0,C 180,E1 -10320.895,E2 -10320.895} C_VEL
LIN {X 0,Y 418.27,Z 548.38,A -85,B 0,C 180,E1 -10324.095,E2 -10324.095} C_VEL
LIN {X 0,Y 418.237,Z 548.385,A -85,B 0,C 180,E1 -10327.263,E2 -10327.263} C_VEL
LIN {X 0,Y 418.282,Z 548.38,A -85,B 0,C 180,E1 -10330.364,E2 -10330.364} C_VEL
LIN {X 0,Y 418.316,Z 548.375,A -85,B 0,C 180,E1 -10333.404,E2 -10333.404} C_VEL
LIN {X 0,Y 418.345,Z 548.376,A -85,B 0,C 180,E1 -10336.999,E2 -10336.999} C_VEL
LIN {X 0,Y 418.34,Z 548.371,A -85,B 0,C 180,E1 -10340.328,E2 -10340.328} C_VEL
LIN {X 0,Y 418.492,Z 548.356,A -85,B 0,C 180,E1 -10343.248,E2 -10343.248} C_VEL
LIN {X 0,Y 418.339,Z 548.376,A -85,B 0,C 180,E1 -10345.181,E2 -10345.181} C_VEL
LIN {X 0,Y 418.543,Z 548.345,A -85,B 0,C 180,E1 -10348.075,E2 -10348.075} C_VEL
LIN {X 0,Y 418.671,Z 548.329,A -85,B 0,C 180,E1 -10349.999,E2 -10349.999} C_VEL
LIN {X 0,Y 418.509,Z 548.353,A -85,B 0,C 180,E1 -10352.887,E2 -10352.887} C_VEL
LIN {X 0,Y 418.288,Z 548.377,A -85,B 0,C 180,E1 -10353.898,E2 -10353.898} C_VEL
LIN {X 0,Y 417.662,Z 548.458,A -85,B 0,C 180,E1 -10354.702,E2 -10354.702} C_VEL
LIN {X 0,Y 414.945,Z 548.793,A -85,B 0,C 180,E1 -10356.013,E2 -10356.013} C_VEL
LIN {X 0,Y 412.602,Z 549.09,A -85,B 0,C 180,E1 -10357.07,E2 -10357.07} C_VEL
LIN {X 0,Y 411.542,Z 549.219,A -85,B 0,C 180,E1 -10357.885,E2 -10357.885} C_VEL
LIN {X 0,Y 411.426,Z 549.231,A -85,B 0,C 180,E1 -10358.162,E2 -10358.162} C_VEL
LIN {X 0,Y 411.298,Z 549.25,A -85,B 0,C 180,E1 -10361.832,E2 -10361.832} C_VEL
LIN {X 0,Y 411.26,Z 549.254,A -85,B 0,C 180,E1 -10364.852,E2 -10364.852} C_VEL
LIN {X 0,Y 411.249,Z 549.256,A -85,B 0,C 180,E1 -10367.915,E2 -10367.915} C_VEL
LIN {X 0,Y 411.193,Z 549.262,A -85,B 0,C 180,E1 -10371.034,E2 -10371.034} C_VEL
LIN {X 0,Y 411.223,Z 549.258,A -85,B 0,C 180,E1 -10374.215,E2 -10374.215} C_VEL
LIN {X 0,Y 411.255,Z 549.258,A -85,B 0,C 180,E1 -10377.477,E2 -10377.477} C_VEL
LIN {X 0,Y 411.197,Z 549.26,A -85,B 0,C 180,E1 -10380.846,E2 -10380.846} C_VEL
LIN {X 0,Y 411.201,Z 549.261,A -85,B 0,C 180,E1 -10384.333,E2 -10384.333} C_VEL
LIN {X 0,Y 411.199,Z 549.266,A -85,B 0,C 180,E1 -10387.972,E2 -10387.972} C_VEL
LIN {X 0,Y 411.195,Z 549.261,A -85,B 0,C 180,E1 -10391.234,E2 -10391.234} C_VEL
LIN {X 0,Y 411.181,Z 549.264,A -85,B 0,C 180,E1 -10394.489,E2 -10394.489} C_VEL
LIN {X 0,Y 411.227,Z 549.257,A -85,B 0,C 180,E1 -10397.296,E2 -10397.296} C_VEL
LIN {X 0,Y 411.228,Z 549.257,A -85,B 0,C 180,E1 -10400.778,E2 -10400.778} C_VEL
LIN {X 0,Y 411.195,Z 549.264,A -85,B 0,C 180,E1 -10404.471,E2 -10404.471} C_VEL
LIN {X 0,Y 411.271,Z 549.361,A -85,B 0,C 180,E1 -10405.747,E2 -10405.747} C_VEL
LIN {X 0,Y 417.829,Z 567.311,A -85,B 0,C 180,E1 -10406.394,E2 -10406.394} C_VEL
LIN {X 0,Y 417.311,Z 609.198,A -85,B 0,C 180,E1 -10407.225,E2 -10407.225} C_VEL
LIN {X 0,Y 417.103,Z 623.313,A -85,B 0,C 180,E1 -10407.694,E2 -10407.694} C_VEL
LIN {X 0,Y 416.714,Z 636.884,A -85,B 0,C 180,E1 -10408.337,E2 -10408.337} C_VEL
LIN {X 0,Y 416.145,Z 650.405,A -85,B 0,C 180,E1 -10409.193,E2 -10409.193} C_VEL
LIN {X 0,Y 415.519,Z 663.008,A -85,B 0,C 180,E1 -10410.209,E2 -10410.209} C_VEL
LIN {X 0,Y 414.751,Z 674.969,A -85,B 0,C 180,E1 -10411.4,E2 -10411.4} C_VEL
LIN {X 0,Y 414.016,Z 685.808,A -85,B 0,C 180,E1 -10412.721,E2 -10412.721} C_VEL
LIN {X 0,Y 413.351,Z 695.454,A -85,B 0,C 180,E1 -10414.157,E2 -10414.157} C_VEL
LIN {X 0,Y 412.738,Z 703.573,A -85,B 0,C 180,E1 -10415.612,E2 -10415.612} C_VEL
LIN {X 0,Y 412.267,Z 710.075,A -85,B 0,C 180,E1 -10417.004,E2 -10417.004} C_VEL
LIN {X 0,Y 411.849,Z 715.773,A -85,B 0,C 180,E1 -10418.477,E2 -10418.477} C_VEL
LIN {X 0,Y 411.546,Z 720.643,A -85,B 0,C 180,E1 -10420.03,E2 -10420.03} C_VEL
LIN {X 0,Y 411.302,Z 724.457,A -85,B 0,C 180,E1 -10421.572,E2 -10421.572} C_VEL
LIN {X 0,Y 411.113,Z 727.47,A -85,B 0,C 180,E1 -10423.198,E2 -10423.198} C_VEL
LIN {X 0,Y 410.995,Z 729.792,A -85,B 0,C 180,E1 -10425.138,E2 -10425.138} C_VEL
LIN {X 0,Y 411.049,Z 730.794,A -85,B 0,C 180,E1 -10427.158,E2 -10427.158} C_VEL
LIN {X 0,Y 411.116,Z 730.328,A -85,B 0,C 180,E1 -10429.162,E2 -10429.162} C_VEL
LIN {X 0,Y 411.333,Z 728.434,A -85,B 0,C 180,E1 -10431.155,E2 -10431.155} C_VEL
LIN {X 0,Y 411.72,Z 725.096,A -85,B 0,C 180,E1 -10433.138,E2 -10433.138} C_VEL
LIN {X 0,Y 412.039,Z 721.575,A -85,B 0,C 180,E1 -10434.618,E2 -10434.618} C_VEL
LIN {X 0,Y 412.441,Z 717.134,A -85,B 0,C 180,E1 -10436.092,E2 -10436.092} C_VEL
LIN {X 0,Y 413.124,Z 710.593,A -85,B 0,C 180,E1 -10437.807,E2 -10437.807} C_VEL
LIN {X 0,Y 413.823,Z 702.459,A -85,B 0,C 180,E1 -10439.514,E2 -10439.514} C_VEL
LIN {X 0,Y 414.712,Z 693.546,A -85,B 0,C 180,E1 -10441.021,E2 -10441.021} C_VEL
LIN {X 0,Y 415.433,Z 683.407,A -85,B 0,C 180,E1 -10442.424,E2 -10442.424} C_VEL
LIN {X 0,Y 416.158,Z 674.239,A -85,B 0,C 180,E1 -10443.473,E2 -10443.473} C_VEL
LIN {X 0,Y 416.946,Z 662.291,A -85,B 0,C 180,E1 -10444.593,E2 -10444.593} C_VEL
LIN {X 0,Y 417.619,Z 649.39,A -85,B 0,C 180,E1 -10445.553,E2 -10445.553} C_VEL
LIN {X 0,Y 418.05,Z 636.323,A -85,B 0,C 180,E1 -10446.308,E2 -10446.308} C_VEL
LIN {X 0,Y 418.317,Z 622.604,A -85,B 0,C 180,E1 -10446.882,E2 -10446.882} C_VEL
LIN {X 0,Y 418.329,Z 607.836,A -85,B 0,C 180,E1 -10447.287,E2 -10447.287} C_VEL
LIN {X 0,Y 418.798,Z 566.841,A -85,B 0,C 180,E1 -10448.074,E2 -10448.074} C_VEL
LIN {X 0,Y 413.567,Z 554.638,A -85,B 0,C 180,E1 -10448.654,E2 -10448.654} C_VEL
LIN {X 0,Y 411.43,Z 549.705,A -85,B 0,C 180,E1 -10448.906,E2 -10448.906} C_VEL
LIN {X 0,Y 411.339,Z 549.249,A -85,B 0,C 180,E1 -10448.939,E2 -10448.939} C_VEL
LIN {X 0,Y 411.295,Z 549.256,A -85,B 0,C 180,E1 -10451.833,E2 -10451.833} C_VEL
LIN {X 0,Y 411.259,Z 549.26,A -85,B 0,C 180,E1 -10454.853,E2 -10454.853} C_VEL
LIN {X 0,Y 411.249,Z 549.26,A -85,B 0,C 180,E1 -10457.916,E2 -10457.916} C_VEL
LIN {X 0,Y 411.194,Z 549.267,A -85,B 0,C 180,E1 -10461.035,E2 -10461.035} C_VEL
LIN {X 0,Y 411.224,Z 549.26,A -85,B 0,C 180,E1 -10464.216,E2 -10464.216} C_VEL
LIN {X 0,Y 411.257,Z 549.253,A -85,B 0,C 180,E1 -10467.478,E2 -10467.478} C_VEL
LIN {X 0,Y 411.196,Z 549.258,A -85,B 0,C 180,E1 -10470.848,E2 -10470.848} C_VEL
LIN {X 0,Y 411.203,Z 549.255,A -85,B 0,C 180,E1 -10474.334,E2 -10474.334} C_VEL
LIN {X 0,Y 411.199,Z 549.261,A -85,B 0,C 180,E1 -10477.974,E2 -10477.974} C_VEL
LIN {X 0,Y 411.182,Z 549.263,A -85,B 0,C 180,E1 -10480.505,E2 -10480.505} C_VEL
LIN {X 0,Y 411.176,Z 549.269,A -85,B 0,C 180,E1 -10483.134,E2 -10483.134} C_VEL
LIN {X 0,Y 411.167,Z 549.265,A -85,B 0,C 180,E1 -10485.882,E2 -10485.882} C_VEL
LIN {X 0,Y 411.163,Z 549.263,A -85,B 0,C 180,E1 -10488.772,E2 -10488.772} C_VEL
LIN {X 0,Y 411.21,Z 549.265,A -85,B 0,C 180,E1 -10491.831,E2 -10491.831} C_VEL
LIN {X 0,Y 411.22,Z 549.43,A -85,B 0,C 180,E1 -10493.262,E2 -10493.262} C_VEL
LIN {X 0,Y 414.361,Z 563.991,A -85,B 0,C 180,E1 -10496.594,E2 -10496.594} C_VEL
LIN {X 0,Y 415.728,Z 570.723,A -85,B 0,C 180,E1 -10498.083,E2 -10498.083} C_VEL
LIN {X 0,Y 414.991,Z 581.7,A -85,B 0,C 180,E1 -10500.318,E2 -10500.318} C_VEL
LIN {X 0,Y 413.696,Z 599.057,A -85,B 0,C 180,E1 -10503.789,E2 -10503.789} C_VEL
LIN {X 0,Y 412.652,Z 616.392,A -85,B 0,C 180,E1 -10507.204,E2 -10507.204} C_VEL
LIN {X 0,Y 411.966,Z 630.161,A -85,B 0,C 180,E1 -10509.89,E2 -10509.89} C_VEL
LIN {X 0,Y 417.307,Z 674.036,A -85,B 0,C 180,E1 -10511.179,E2 -10511.179} C_VEL
LIN {X 0,Y 415.621,Z 744.561,A -85,B 0,C 180,E1 -10512.788,E2 -10512.788} C_VEL
LIN {X 0,Y 415.013,Z 757.771,A -85,B 0,C 180,E1 -10513.269,E2 -10513.269} C_VEL
LIN {X 0,Y 414.185,Z 770.73,A -85,B 0,C 180,E1 -10513.932,E2 -10513.932} C_VEL
LIN {X 0,Y 413.389,Z 782.393,A -85,B 0,C 180,E1 -10514.722,E2 -10514.722} C_VEL
LIN {X 0,Y 412.638,Z 793.848,A -85,B 0,C 180,E1 -10515.703,E2 -10515.703} C_VEL
LIN {X 0,Y 411.899,Z 804.777,A -85,B 0,C 180,E1 -10516.859,E2 -10516.859} C_VEL
LIN {X 0,Y 411.333,Z 813.034,A -85,B 0,C 180,E1 -10517.919,E2 -10517.919} C_VEL
LIN {X 0,Y 410.902,Z 821.123,A -85,B 0,C 180,E1 -10519.156,E2 -10519.156} C_VEL
LIN {X 0,Y 410.603,Z 829.084,A -85,B 0,C 180,E1 -10520.643,E2 -10520.643} C_VEL
LIN {X 0,Y 410.471,Z 835.483,A -85,B 0,C 180,E1 -10522.128,E2 -10522.128} C_VEL
LIN {X 0,Y 410.482,Z 840.477,A -85,B 0,C 180,E1 -10523.584,E2 -10523.584} C_VEL
LIN {X 0,Y 410.545,Z 844.438,A -85,B 0,C 180,E1 -10525.09,E2 -10525.09} C_VEL
LIN {X 0,Y 410.612,Z 846.412,A -85,B 0,C 180,E1 -10526.075,E2 -10526.075} C_VEL
LIN {X 0,Y 410.578,Z 847.917,A -85,B 0,C 180,E1 -10527.057,E2 -10527.057} C_VEL
LIN {X 0,Y 410.593,Z 848.938,A -85,B 0,C 180,E1 -10528.039,E2 -10528.039} C_VEL
LIN {X 0,Y 410.616,Z 849.51,A -85,B 0,C 180,E1 -10529.02,E2 -10529.02} C_VEL
LIN {X 0,Y 410.849,Z 849.68,A -85,B 0,C 180,E1 -10530.001,E2 -10530.001} C_VEL
LIN {X 0,Y 410.636,Z 849.354,A -85,B 0,C 180,E1 -10530.981,E2 -10530.981} C_VEL
LIN {X 0,Y 410.632,Z 848.584,A -85,B 0,C 180,E1 -10531.962,E2 -10531.962} C_VEL
LIN {X 0,Y 410.631,Z 847.361,A -85,B 0,C 180,E1 -10532.944,E2 -10532.944} C_VEL
LIN {X 0,Y 410.676,Z 844.696,A -85,B 0,C 180,E1 -10534.417,E2 -10534.417} C_VEL
LIN {X 0,Y 410.538,Z 840.92,A -85,B 0,C 180,E1 -10535.896,E2 -10535.896} C_VEL
LIN {X 0,Y 410.519,Z 835.975,A -85,B 0,C 180,E1 -10537.378,E2 -10537.378} C_VEL
LIN {X 0,Y 410.573,Z 829.742,A -85,B 0,C 180,E1 -10538.863,E2 -10538.863} C_VEL
LIN {X 0,Y 410.761,Z 822.046,A -85,B 0,C 180,E1 -10540.35,E2 -10540.35} C_VEL
LIN {X 0,Y 411.176,Z 812.611,A -85,B 0,C 180,E1 -10541.836,E2 -10541.836} C_VEL
LIN {X 0,Y 411.574,Z 803.944,A -85,B 0,C 180,E1 -10542.968,E2 -10542.968} C_VEL
LIN {X 0,Y 412.431,Z 792.705,A -85,B 0,C 180,E1 -10544.18,E2 -10544.18} C_VEL
LIN {X 0,Y 412.929,Z 784.608,A -85,B 0,C 180,E1 -10544.918,E2 -10544.918} C_VEL
LIN {X 0,Y 413.953,Z 771.638,A -85,B 0,C 180,E1 -10545.889,E2 -10545.889} C_VEL
LIN {X 0,Y 414.869,Z 758.207,A -85,B 0,C 180,E1 -10546.675,E2 -10546.675} C_VEL
LIN {X 0,Y 415.744,Z 744.466,A -85,B 0,C 180,E1 -10547.271,E2 -10547.271} C_VEL
LIN {X 0,Y 416.316,Z 729.233,A -85,B 0,C 180,E1 -10547.722,E2 -10547.722} C_VEL
LIN {X 0,Y 417.555,Z 673.046,A -85,B 0,C 180,E1 -10548.957,E2 -10548.957} C_VEL
LIN {X 0,Y 416.256,Z 655.224,A -85,B 0,C 180,E1 -10549.466,E2 -10549.466} C_VEL
LIN {X 0,Y 414.713,Z 634.417,A -85,B 0,C 180,E1 -10550.084,E2 -10550.084} C_VEL
LIN {X 0,Y 412.031,Z 613.947,A -85,B 0,C 180,E1 -10550.797,E2 -10550.797} C_VEL
LIN {X 0,Y 411.521,Z 609.91,A -85,B 0,C 180,E1 -10550.953,E2 -10550.953} C_VEL
LIN {X 0,Y 411.825,Z 590.695,A -85,B 0,C 180,E1 -10554.447,E2 -10554.447} C_VEL
LIN {X 0,Y 412.302,Z 571.787,A -85,B 0,C 180,E1 -10557.981,E2 -10557.981} C_VEL
LIN {X 0,Y 412.768,Z 559.063,A -85,B 0,C 180,E1 -10560.434,E2 -10560.434} C_VEL
LIN {X 0,Y 411.752,Z 551.727,A -85,B 0,C 180,E1 -10561.947,E2 -10561.947} C_VEL
LIN {X 0,Y 411.243,Z 549.264,A -85,B 0,C 180,E1 -10562.498,E2 -10562.498} C_VEL
LIN {X 0,Y 411.203,Z 549.263,A -85,B 0,C 180,E1 -10565.529,E2 -10565.529} C_VEL
LIN {X 0,Y 411.222,Z 549.262,A -85,B 0,C 180,E1 -10569.224,E2 -10569.224} C_VEL
LIN {X 0,Y 411.186,Z 549.266,A -85,B 0,C 180,E1 -10572.696,E2 -10572.696} C_VEL
LIN {X 0,Y 411.173,Z 549.266,A -85,B 0,C 180,E1 -10575.881,E2 -10575.881} C_VEL
LIN {X 0,Y 411.168,Z 549.268,A -85,B 0,C 180,E1 -10578.772,E2 -10578.772} C_VEL
LIN {X 0,Y 411.211,Z 549.262,A -85,B 0,C 180,E1 -10581.831,E2 -10581.831} C_VEL
LIN {X 0,Y 411.215,Z 549.263,A -85,B 0,C 180,E1 -10585.121,E2 -10585.121} C_VEL
LIN {X 0,Y 411.17,Z 549.267,A -85,B 0,C 180,E1 -10588.003,E2 -10588.003} C_VEL
LIN {X 0,Y 411.223,Z 549.262,A -85,B 0,C 180,E1 -10591.41,E2 -10591.41} C_VEL
LIN {X 0,Y 411.243,Z 549.262,A -85,B 0,C 180,E1 -10593.619,E2 -10593.619} C_VEL
LIN {X 0,Y 411.208,Z 549.266,A -85,B 0,C 180,E1 -10596.852,E2 -10596.852} C_VEL
LIN {X 0,Y 411.229,Z 549.384,A -85,B 0,C 180,E1 -10598.585,E2 -10598.585} C_VEL
LIN {X 0,Y 412.248,Z 552.124,A -85,B 0,C 180,E1 -10598.717,E2 -10598.717} C_VEL
LIN {X 0,Y 418.391,Z 564.898,A -85,B 0,C 180,E1 -10599.42,E2 -10599.42} C_VEL
LIN {X 0,Y 420.008,Z 568.795,A -85,B 0,C 180,E1 -10599.601,E2 -10599.601} C_VEL
LIN {X 0,Y 419.97,Z 600.501,A -85,B 0,C 180,E1 -10600.222,E2 -10600.222} C_VEL
LIN {X 0,Y 419.947,Z 614.983,A -85,B 0,C 180,E1 -10600.676,E2 -10600.676} C_VEL
LIN {X 0,Y 419.706,Z 629.402,A -85,B 0,C 180,E1 -10601.328,E2 -10601.328} C_VEL
LIN {X 0,Y 419.161,Z 643.572,A -85,B 0,C 180,E1 -10602.182,E2 -10602.182} C_VEL
LIN {X 0,Y 418.491,Z 656.688,A -85,B 0,C 180,E1 -10603.185,E2 -10603.185} C_VEL
LIN {X 0,Y 417.736,Z 667.835,A -85,B 0,C 180,E1 -10604.221,E2 -10604.221} C_VEL
LIN {X 0,Y 416.951,Z 677.959,A -85,B 0,C 180,E1 -10605.354,E2 -10605.354} C_VEL
LIN {X 0,Y 415.955,Z 688.895,A -85,B 0,C 180,E1 -10606.815,E2 -10606.815} C_VEL
LIN {X 0,Y 414.953,Z 699.304,A -85,B 0,C 180,E1 -10608.521,E2 -10608.521} C_VEL
LIN {X 0,Y 414.07,Z 707.814,A -85,B 0,C 180,E1 -10610.227,E2 -10610.227} C_VEL
LIN {X 0,Y 413.443,Z 713.867,A -85,B 0,C 180,E1 -10611.692,E2 -10611.692} C_VEL
LIN {X 0,Y 412.722,Z 718.956,A -85,B 0,C 180,E1 -10613.154,E2 -10613.154} C_VEL
LIN {X 0,Y 412.425,Z 723.134,A -85,B 0,C 180,E1 -10614.622,E2 -10614.622} C_VEL
LIN {X 0,Y 412.059,Z 726.462,A -85,B 0,C 180,E1 -10616.088,E2 -10616.088} C_VEL
LIN {X 0,Y 411.641,Z 729.784,A -85,B 0,C 180,E1 -10618.043,E2 -10618.043} C_VEL
LIN {X 0,Y 411.366,Z 731.85,A -85,B 0,C 180,E1 -10620,E2 -10620} C_VEL
LIN {X 0,Y 411.296,Z 732.702,A -85,B 0,C 180,E1 -10621.958,E2 -10621.958} C_VEL
LIN {X 0,Y 411.095,Z 732.388,A -85,B 0,C 180,E1 -10623.921,E2 -10623.921} C_VEL
LIN {X 0,Y 411.334,Z 730.822,A -85,B 0,C 180,E1 -10625.884,E2 -10625.884} C_VEL
LIN {X 0,Y 411.378,Z 728.055,A -85,B 0,C 180,E1 -10627.855,E2 -10627.855} C_VEL
LIN {X 0,Y 411.621,Z 723.973,A -85,B 0,C 180,E1 -10629.83,E2 -10629.83} C_VEL
LIN {X 0,Y 411.907,Z 718.497,A -85,B 0,C 180,E1 -10631.814,E2 -10631.814} C_VEL
LIN {X 0,Y 412.452,Z 711.423,A -85,B 0,C 180,E1 -10633.801,E2 -10633.801} C_VEL
LIN {X 0,Y 413.058,Z 703.755,A -85,B 0,C 180,E1 -10635.544,E2 -10635.544} C_VEL
LIN {X 0,Y 413.751,Z 694.411,A -85,B 0,C 180,E1 -10637.292,E2 -10637.292} C_VEL
LIN {X 0,Y 414.494,Z 684.81,A -85,B 0,C 180,E1 -10638.793,E2 -10638.793} C_VEL
LIN {X 0,Y 415.346,Z 673.261,A -85,B 0,C 180,E1 -10640.296,E2 -10640.296} C_VEL
LIN {X 0,Y 416.198,Z 661.023,A -85,B 0,C 180,E1 -10641.617,E2 -10641.617} C_VEL
LIN {X 0,Y 416.879,Z 649.216,A -85,B 0,C 180,E1 -10642.683,E2 -10642.683} C_VEL
LIN {X 0,Y 417.602,Z 635.527,A -85,B 0,C 180,E1 -10643.69,E2 -10643.69} C_VEL
LIN {X 0,Y 418.19,Z 621.454,A -85,B 0,C 180,E1 -10644.512,E2 -10644.512} C_VEL
LIN {X 0,Y 418.619,Z 606.455,A -85,B 0,C 180,E1 -10645.176,E2 -10645.176} C_VEL
LIN {X 0,Y 418.78,Z 592.09,A -85,B 0,C 180,E1 -10645.631,E2 -10645.631} C_VEL
LIN {X 0,Y 418.937,Z 569.94,A -85,B 0,C 180,E1 -10646.094,E2 -10646.094} C_VEL
LIN {X 0,Y 411.317,Z 549.598,A -85,B 0,C 180,E1 -10646.865,E2 -10646.865} C_VEL
LIN {X 0,Y 411.29,Z 549.252,A -85,B 0,C 180,E1 -10646.911,E2 -10646.911} C_VEL
LIN {X 0,Y 411.202,Z 549.265,A -85,B 0,C 180,E1 -10649.712,E2 -10649.712} C_VEL
LIN {X 0,Y 411.207,Z 549.259,A -85,B 0,C 180,E1 -10653.155,E2 -10653.155} C_VEL
LIN {X 0,Y 411.193,Z 549.263,A -85,B 0,C 180,E1 -10656.552,E2 -10656.552} C_VEL
LIN {X 0,Y 411.213,Z 549.26,A -85,B 0,C 180,E1 -10659.727,E2 -10659.727} C_VEL
LIN {X 0,Y 411.173,Z 549.263,A -85,B 0,C 180,E1 -10663.133,E2 -10663.133} C_VEL
LIN {X 0,Y 411.168,Z 549.266,A -85,B 0,C 180,E1 -10665.88,E2 -10665.88} C_VEL
LIN {X 0,Y 411.165,Z 549.267,A -85,B 0,C 180,E1 -10668.771,E2 -10668.771} C_VEL
LIN {X 0,Y 411.211,Z 549.259,A -85,B 0,C 180,E1 -10671.83,E2 -10671.83} C_VEL
LIN {X 0,Y 411.211,Z 549.259,A -85,B 0,C 180,E1 -10675.121,E2 -10675.121} C_VEL
LIN {X 0,Y 411.165,Z 549.265,A -85,B 0,C 180,E1 -10678.002,E2 -10678.002} C_VEL
LIN {X 0,Y 411.217,Z 549.258,A -85,B 0,C 180,E1 -10681.409,E2 -10681.409} C_VEL
LIN {X 0,Y 411.237,Z 549.255,A -85,B 0,C 180,E1 -10683.619,E2 -10683.619} C_VEL
LIN {X 0,Y 411.202,Z 549.265,A -85,B 0,C 180,E1 -10686.852,E2 -10686.852} C_VEL
LIN {X 0,Y 411.214,Z 549.258,A -85,B 0,C 180,E1 -10690.05,E2 -10690.05} C_VEL
LIN {X 0,Y 411.262,Z 549.256,A -85,B 0,C 180,E1 -10693.131,E2 -10693.131} C_VEL
LIN {X 0,Y 411.304,Z 549.255,A -85,B 0,C 180,E1 -10696.895,E2 -10696.895} C_VEL
LIN {X 0,Y 411.292,Z 549.248,A -85,B 0,C 180,E1 -10700.161,E2 -10700.161} C_VEL
LIN {X 0,Y 411.459,Z 549.234,A -85,B 0,C 180,E1 -10703.132,E2 -10703.132} C_VEL
LIN {X 0,Y 411.31,Z 549.253,A -85,B 0,C 180,E1 -10705.098,E2 -10705.098} C_VEL
LIN {X 0,Y 411.512,Z 549.221,A -85,B 0,C 180,E1 -10708.042,E2 -10708.042} C_VEL
LIN {X 0,Y 411.64,Z 549.205,A -85,B 0,C 180,E1 -10709.999,E2 -10709.999} C_VEL
LIN {X 0,Y 411.465,Z 549.231,A -85,B 0,C 180,E1 -10712.937,E2 -10712.937} C_VEL
LIN {X 0,Y 411.452,Z 549.231,A -85,B 0,C 180,E1 -10716.866,E2 -10716.866} C_VEL
LIN {X 0,Y 411.426,Z 549.231,A -85,B 0,C 180,E1 -10718.162,E2 -10718.162} C_VEL
LIN {X 0,Y 410.672,Z 549.331,A -85,B 0,C 180,E1 -10718.978,E2 -10718.978} C_VEL
LIN {X 0,Y 407.765,Z 549.687,A -85,B 0,C 180,E1 -10720.305,E2 -10720.305} C_VEL
LIN {X 0,Y 405.358,Z 549.995,A -85,B 0,C 180,E1 -10721.376,E2 -10721.376} C_VEL
LIN {X 0,Y 404.337,Z 550.115,A -85,B 0,C 180,E1 -10722.205,E2 -10722.205} C_VEL
LIN {X 0,Y 404.257,Z 550.124,A -85,B 0,C 180,E1 -10722.485,E2 -10722.485} C_VEL
LIN {X 0,Y 404.218,Z 550.13,A -85,B 0,C 180,E1 -10726.151,E2 -10726.151} C_VEL
LIN {X 0,Y 404.162,Z 550.141,A -85,B 0,C 180,E1 -10729.292,E2 -10729.292} C_VEL
LIN {X 0,Y 404.152,Z 550.138,A -85,B 0,C 180,E1 -10732.834,E2 -10732.834} C_VEL
LIN {X 0,Y 404.179,Z 550.14,A -85,B 0,C 180,E1 -10735.766,E2 -10735.766} C_VEL
LIN {X 0,Y 404.193,Z 550.136,A -85,B 0,C 180,E1 -10737.999,E2 -10737.999} C_VEL
LIN {X 0,Y 404.146,Z 550.142,A -85,B 0,C 180,E1 -10741.445,E2 -10741.445} C_VEL
LIN {X 0,Y 404.181,Z 550.134,A -85,B 0,C 180,E1 -10745.016,E2 -10745.016} C_VEL
LIN {X 0,Y 404.158,Z 550.137,A -85,B 0,C 180,E1 -10748.756,E2 -10748.756} C_VEL
LIN {X 0,Y 404.144,Z 550.142,A -85,B 0,C 180,E1 -10751.604,E2 -10751.604} C_VEL
LIN {X 0,Y 404.149,Z 550.139,A -85,B 0,C 180,E1 -10754.523,E2 -10754.523} C_VEL
LIN {X 0,Y 404.205,Z 550.132,A -85,B 0,C 180,E1 -10757.305,E2 -10757.305} C_VEL
LIN {X 0,Y 404.165,Z 550.142,A -85,B 0,C 180,E1 -10759.956,E2 -10759.956} C_VEL
LIN {X 0,Y 404.136,Z 550.14,A -85,B 0,C 180,E1 -10763.124,E2 -10763.124} C_VEL
LIN {X 0,Y 404.19,Z 550.133,A -85,B 0,C 180,E1 -10765.434,E2 -10765.434} C_VEL
LIN {X 0,Y 411.067,Z 568.992,A -85,B 0,C 180,E1 -10766.139,E2 -10766.139} C_VEL
LIN {X 0,Y 410.481,Z 610.276,A -85,B 0,C 180,E1 -10766.977,E2 -10766.977} C_VEL
LIN {X 0,Y 410.295,Z 624.116,A -85,B 0,C 180,E1 -10767.445,E2 -10767.445} C_VEL
LIN {X 0,Y 409.874,Z 637.918,A -85,B 0,C 180,E1 -10768.108,E2 -10768.108} C_VEL
LIN {X 0,Y 409.267,Z 651.635,A -85,B 0,C 180,E1 -10768.992,E2 -10768.992} C_VEL
LIN {X 0,Y 408.588,Z 664.785,A -85,B 0,C 180,E1 -10770.079,E2 -10770.079} C_VEL
LIN {X 0,Y 407.798,Z 676.755,A -85,B 0,C 180,E1 -10771.303,E2 -10771.303} C_VEL
LIN {X 0,Y 407.117,Z 686.356,A -85,B 0,C 180,E1 -10772.498,E2 -10772.498} C_VEL
LIN {X 0,Y 406.532,Z 694.824,A -85,B 0,C 180,E1 -10773.752,E2 -10773.752} C_VEL
LIN {X 0,Y 405.871,Z 702.933,A -85,B 0,C 180,E1 -10775.172,E2 -10775.172} C_VEL
LIN {X 0,Y 405.317,Z 710.526,A -85,B 0,C 180,E1 -10776.778,E2 -10776.778} C_VEL
LIN {X 0,Y 404.792,Z 717.508,A -85,B 0,C 180,E1 -10778.617,E2 -10778.617} C_VEL
LIN {X 0,Y 404.505,Z 722.337,A -85,B 0,C 180,E1 -10780.224,E2 -10780.224} C_VEL
LIN {X 0,Y 404.242,Z 725.959,A -85,B 0,C 180,E1 -10781.764,E2 -10781.764} C_VEL
LIN {X 0,Y 404.1,Z 728.268,A -85,B 0,C 180,E1 -10783.045,E2 -10783.045} C_VEL
LIN {X 0,Y 403.964,Z 730.569,A -85,B 0,C 180,E1 -10784.873,E2 -10784.873} C_VEL
LIN {X 0,Y 404.027,Z 731.761,A -85,B 0,C 180,E1 -10786.931,E2 -10786.931} C_VEL
LIN {X 0,Y 404.109,Z 731.537,A -85,B 0,C 180,E1 -10788.972,E2 -10788.972} C_VEL
LIN {X 0,Y 404.329,Z 729.845,A -85,B 0,C 180,E1 -10791,E2 -10791} C_VEL
LIN {X 0,Y 404.7,Z 726.684,A -85,B 0,C 180,E1 -10793.018,E2 -10793.018} C_VEL
LIN {X 0,Y 405.174,Z 722.016,A -85,B 0,C 180,E1 -10795.025,E2 -10795.025} C_VEL
LIN {X 0,Y 405.645,Z 717.405,A -85,B 0,C 180,E1 -10796.524,E2 -10796.524} C_VEL
LIN {X 0,Y 406.336,Z 710.71,A -85,B 0,C 180,E1 -10798.266,E2 -10798.266} C_VEL
LIN {X 0,Y 407.169,Z 702.303,A -85,B 0,C 180,E1 -10800,E2 -10800} C_VEL
LIN {X 0,Y 408.094,Z 693.379,A -85,B 0,C 180,E1 -10801.481,E2 -10801.481} C_VEL
LIN {X 0,Y 408.74,Z 684.537,A -85,B 0,C 180,E1 -10802.711,E2 -10802.711} C_VEL
LIN {X 0,Y 409.655,Z 673.763,A -85,B 0,C 180,E1 -10803.935,E2 -10803.935} C_VEL
LIN {X 0,Y 410.407,Z 661.92,A -85,B 0,C 180,E1 -10805.035,E2 -10805.035} C_VEL
LIN {X 0,Y 411.086,Z 648.677,A -85,B 0,C 180,E1 -10806.011,E2 -10806.011} C_VEL
LIN {X 0,Y 411.525,Z 635.605,A -85,B 0,C 180,E1 -10806.743,E2 -10806.743} C_VEL
LIN {X 0,Y 411.759,Z 621.17,A -85,B 0,C 180,E1 -10807.327,E2 -10807.327} C_VEL
LIN {X 0,Y 411.811,Z 606.906,A -85,B 0,C 180,E1 -10807.692,E2 -10807.692} C_VEL
LIN {X 0,Y 412.284,Z 568.609,A -85,B 0,C 180,E1 -10808.444,E2 -10808.444} C_VEL
LIN {X 0,Y 407.006,Z 556.365,A -85,B 0,C 180,E1 -10809.059,E2 -10809.059} C_VEL
LIN {X 0,Y 404.401,Z 550.724,A -85,B 0,C 180,E1 -10809.368,E2 -10809.368} C_VEL
LIN {X 0,Y 404.313,Z 550.124,A -85,B 0,C 180,E1 -10809.417,E2 -10809.417} C_VEL
LIN {X 0,Y 404.263,Z 550.134,A -85,B 0,C 180,E1 -10813.212,E2 -10813.212} C_VEL
LIN {X 0,Y 404.212,Z 550.137,A -85,B 0,C 180,E1 -10817.008,E2 -10817.008} C_VEL
LIN {X 0,Y 404.161,Z 550.141,A -85,B 0,C 180,E1 -10820.352,E2 -10820.352} C_VEL
LIN {X 0,Y 404.167,Z 550.14,A -85,B 0,C 180,E1 -10823.575,E2 -10823.575} C_VEL
LIN {X 0,Y 404.181,Z 550.136,A -85,B 0,C 180,E1 -10825.767,E2 -10825.767} C_VEL
LIN {X 0,Y 404.195,Z 550.132,A -85,B 0,C 180,E1 -10828,E2 -10828} C_VEL
LIN {X 0,Y 404.141,Z 550.137,A -85,B 0,C 180,E1 -10831.56,E2 -10831.56} C_VEL
LIN {X 0,Y 404.183,Z 550.131,A -85,B 0,C 180,E1 -10835.017,E2 -10835.017} C_VEL
LIN {X 0,Y 404.157,Z 550.139,A -85,B 0,C 180,E1 -10838.757,E2 -10838.757} C_VEL
LIN {X 0,Y 404.123,Z 550.142,A -85,B 0,C 180,E1 -10841.601,E2 -10841.601} C_VEL
LIN {X 0,Y 404.147,Z 550.14,A -85,B 0,C 180,E1 -10844.523,E2 -10844.523} C_VEL
LIN {X 0,Y 404.135,Z 550.145,A -85,B 0,C 180,E1 -10847.296,E2 -10847.296} C_VEL
LIN {X 0,Y 404.168,Z 550.139,A -85,B 0,C 180,E1 -10849.956,E2 -10849.956} C_VEL
LIN {X 0,Y 404.207,Z 550.245,A -85,B 0,C 180,E1 -10852.993,E2 -10852.993} C_VEL
LIN {X 0,Y 407.397,Z 565.247,A -85,B 0,C 180,E1 -10856.494,E2 -10856.494} C_VEL
LIN {X 0,Y 408.775,Z 572.368,A -85,B 0,C 180,E1 -10858.085,E2 -10858.085} C_VEL
LIN {X 0,Y 407.722,Z 585.779,A -85,B 0,C 180,E1 -10860.86,E2 -10860.86} C_VEL
LIN {X 0,Y 406.393,Z 604.484,A -85,B 0,C 180,E1 -10864.659,E2 -10864.659} C_VEL
LIN {X 0,Y 405.351,Z 621.75,A -85,B 0,C 180,E1 -10868.114,E2 -10868.114} C_VEL
LIN {X 0,Y 404.987,Z 628.914,A -85,B 0,C 180,E1 -10869.534,E2 -10869.534} C_VEL
LIN {X 0,Y 410.5,Z 675.003,A -85,B 0,C 180,E1 -10870.921,E2 -10870.921} C_VEL
LIN {X 0,Y 408.759,Z 743.229,A -85,B 0,C 180,E1 -10872.522,E2 -10872.522} C_VEL
LIN {X 0,Y 408.113,Z 757.136,A -85,B 0,C 180,E1 -10873.042,E2 -10873.042} C_VEL
LIN {X 0,Y 407.258,Z 769.944,A -85,B 0,C 180,E1 -10873.715,E2 -10873.715} C_VEL
LIN {X 0,Y 406.381,Z 782.304,A -85,B 0,C 180,E1 -10874.58,E2 -10874.58} C_VEL
LIN {X 0,Y 405.602,Z 793.588,A -85,B 0,C 180,E1 -10875.578,E2 -10875.578} C_VEL
LIN {X 0,Y 404.829,Z 804.51,A -85,B 0,C 180,E1 -10876.769,E2 -10876.769} C_VEL
LIN {X 0,Y 404.214,Z 813.411,A -85,B 0,C 180,E1 -10877.958,E2 -10877.958} C_VEL
LIN {X 0,Y 403.718,Z 822.656,A -85,B 0,C 180,E1 -10879.469,E2 -10879.469} C_VEL
LIN {X 0,Y 403.489,Z 830.158,A -85,B 0,C 180,E1 -10880.982,E2 -10880.982} C_VEL
LIN {X 0,Y 403.375,Z 836.162,A -85,B 0,C 180,E1 -10882.492,E2 -10882.492} C_VEL
LIN {X 0,Y 403.394,Z 840.867,A -85,B 0,C 180,E1 -10884,E2 -10884} C_VEL
LIN {X 0,Y 403.499,Z 843.338,A -85,B 0,C 180,E1 -10885.004,E2 -10885.004} C_VEL
LIN {X 0,Y 403.575,Z 845.328,A -85,B 0,C 180,E1 -10886.006,E2 -10886.006} C_VEL
LIN {X 0,Y 403.544,Z 846.847,A -85,B 0,C 180,E1 -10887.006,E2 -10887.006} C_VEL
LIN {X 0,Y 403.56,Z 847.896,A -85,B 0,C 180,E1 -10888.005,E2 -10888.005} C_VEL
LIN {X 0,Y 403.588,Z 848.476,A -85,B 0,C 180,E1 -10889.003,E2 -10889.003} C_VEL
LIN {X 0,Y 403.825,Z 848.655,A -85,B 0,C 180,E1 -10890.001,E2 -10890.001} C_VEL
LIN {X 0,Y 403.606,Z 848.33,A -85,B 0,C 180,E1 -10890.998,E2 -10890.998} C_VEL
LIN {X 0,Y 403.593,Z 847.578,A -85,B 0,C 180,E1 -10891.996,E2 -10891.996} C_VEL
LIN {X 0,Y 403.588,Z 846.355,A -85,B 0,C 180,E1 -10892.995,E2 -10892.995} C_VEL
LIN {X 0,Y 403.624,Z 843.691,A -85,B 0,C 180,E1 -10894.495,E2 -10894.495} C_VEL
LIN {X 0,Y 403.479,Z 839.92,A -85,B 0,C 180,E1 -10896,E2 -10896} C_VEL
LIN {X 0,Y 403.465,Z 834.987,A -85,B 0,C 180,E1 -10897.507,E2 -10897.507} C_VEL
LIN {X 0,Y 403.505,Z 827.574,A -85,B 0,C 180,E1 -10899.272,E2 -10899.272} C_VEL
LIN {X 0,Y 403.778,Z 819.653,A -85,B 0,C 180,E1 -10900.785,E2 -10900.785} C_VEL
LIN {X 0,Y 404.149,Z 811.665,A -85,B 0,C 180,E1 -10902.045,E2 -10902.045} C_VEL
LIN {X 0,Y 404.676,Z 801.408,A -85,B 0,C 180,E1 -10903.394,E2 -10903.394} C_VEL
LIN {X 0,Y 405.436,Z 791.918,A -85,B 0,C 180,E1 -10904.43,E2 -10904.43} C_VEL
LIN {X 0,Y 406.298,Z 780.952,A -85,B 0,C 180,E1 -10905.424,E2 -10905.424} C_VEL
LIN {X 0,Y 407.357,Z 767.453,A -85,B 0,C 180,E1 -10906.411,E2 -10906.411} C_VEL
LIN {X 0,Y 408.372,Z 754.533,A -85,B 0,C 180,E1 -10907.141,E2 -10907.141} C_VEL
LIN {X 0,Y 409.322,Z 739.075,A -85,B 0,C 180,E1 -10907.777,E2 -10907.777} C_VEL
LIN {X 0,Y 409.821,Z 723.457,A -85,B 0,C 180,E1 -10908.206,E2 -10908.206} C_VEL
LIN {X 0,Y 410.97,Z 673.55,A -85,B 0,C 180,E1 -10909.339,E2 -10909.339} C_VEL
LIN {X 0,Y 408.488,Z 637.044,A -85,B 0,C 180,E1 -10910.434,E2 -10910.434} C_VEL
LIN {X 0,Y 405.929,Z 616.289,A -85,B 0,C 180,E1 -10911.178,E2 -10911.178} C_VEL
LIN {X 0,Y 404.49,Z 606.922,A -85,B 0,C 180,E1 -10911.568,E2 -10911.568} C_VEL
LIN {X 0,Y 404.843,Z 587.798,A -85,B 0,C 180,E1 -10915.132,E2 -10915.132} C_VEL
LIN {X 0,Y 405.378,Z 570.378,A -85,B 0,C 180,E1 -10918.475,E2 -10918.475} C_VEL
LIN {X 0,Y 405.726,Z 559.011,A -85,B 0,C 180,E1 -10920.731,E2 -10920.731} C_VEL
LIN {X 0,Y 404.208,Z 550.141,A -85,B 0,C 180,E1 -10922.65,E2 -10922.65} C_VEL
LIN {X 0,Y 404.186,Z 550.14,A -85,B 0,C 180,E1 -10925.19,E2 -10925.19} C_VEL
LIN {X 0,Y 404.159,Z 550.142,A -85,B 0,C 180,E1 -10928.757,E2 -10928.757} C_VEL
LIN {X 0,Y 404.127,Z 550.143,A -85,B 0,C 180,E1 -10931.6,E2 -10931.6} C_VEL
LIN {X 0,Y 404.15,Z 550.141,A -85,B 0,C 180,E1 -10934.522,E2 -10934.522} C_VEL
LIN {X 0,Y 404.141,Z 550.144,A -85,B 0,C 180,E1 -10937.296,E2 -10937.296} C_VEL
LIN {X 0,Y 404.173,Z 550.139,A -85,B 0,C 180,E1 -10939.955,E2 -10939.955} C_VEL
LIN {X 0,Y 404.141,Z 550.145,A -85,B 0,C 180,E1 -10943.125,E2 -10943.125} C_VEL
LIN {X 0,Y 404.149,Z 550.142,A -85,B 0,C 180,E1 -10946.188,E2 -10946.188} C_VEL
LIN {X 0,Y 404.15,Z 550.141,A -85,B 0,C 180,E1 -10949.715,E2 -10949.715} C_VEL
LIN {X 0,Y 404.2,Z 550.14,A -85,B 0,C 180,E1 -10953.123,E2 -10953.123} C_VEL
LIN {X 0,Y 404.182,Z 550.141,A -85,B 0,C 180,E1 -10955.334,E2 -10955.334} C_VEL
LIN {X 0,Y 404.186,Z 550.243,A -85,B 0,C 180,E1 -10958.046,E2 -10958.046} C_VEL
LIN {X 0,Y 405.291,Z 553.19,A -85,B 0,C 180,E1 -10958.201,E2 -10958.201} C_VEL
LIN {X 0,Y 411.2,Z 565.038,A -85,B 0,C 180,E1 -10958.902,E2 -10958.902} C_VEL
LIN {X 0,Y 413.621,Z 570.561,A -85,B 0,C 180,E1 -10959.191,E2 -10959.191} C_VEL
LIN {X 0,Y 413.564,Z 603.981,A -85,B 0,C 180,E1 -10959.887,E2 -10959.887} C_VEL
LIN {X 0,Y 413.528,Z 618.695,A -85,B 0,C 180,E1 -10960.387,E2 -10960.387} C_VEL
LIN {X 0,Y 413.166,Z 633.119,A -85,B 0,C 180,E1 -10961.079,E2 -10961.079} C_VEL
LIN {X 0,Y 412.66,Z 646.014,A -85,B 0,C 180,E1 -10961.891,E2 -10961.891} C_VEL
LIN {X 0,Y 411.935,Z 658.891,A -85,B 0,C 180,E1 -10962.91,E2 -10962.91} C_VEL
LIN {X 0,Y 411.02,Z 671.298,A -85,B 0,C 180,E1 -10964.122,E2 -10964.122} C_VEL
LIN {X 0,Y 410.126,Z 681.783,A -85,B 0,C 180,E1 -10965.359,E2 -10965.359} C_VEL
LIN {X 0,Y 409.089,Z 692.274,A -85,B 0,C 180,E1 -10966.842,E2 -10966.842} C_VEL
LIN {X 0,Y 408.214,Z 701,A -85,B 0,C 180,E1 -10968.328,E2 -10968.328} C_VEL
LIN {X 0,Y 407.254,Z 709.416,A -85,B 0,C 180,E1 -10970.062,E2 -10970.062} C_VEL
LIN {X 0,Y 406.594,Z 715.395,A -85,B 0,C 180,E1 -10971.551,E2 -10971.551} C_VEL
LIN {X 0,Y 405.825,Z 720.399,A -85,B 0,C 180,E1 -10973.037,E2 -10973.037} C_VEL
LIN {X 0,Y 405.51,Z 724.53,A -85,B 0,C 180,E1 -10974.53,E2 -10974.53} C_VEL
LIN {X 0,Y 405.118,Z 727.802,A -85,B 0,C 180,E1 -10976.02,E2 -10976.02} C_VEL
LIN {X 0,Y 404.661,Z 731.054,A -85,B 0,C 180,E1 -10978.009,E2 -10978.009} C_VEL
LIN {X 0,Y 404.386,Z 733.038,A -85,B 0,C 180,E1 -10980,E2 -10980} C_VEL
LIN {X 0,Y 404.283,Z 733.801,A -85,B 0,C 180,E1 -10981.992,E2 -10981.992} C_VEL
LIN {X 0,Y 404.072,Z 733.391,A -85,B 0,C 180,E1 -10983.989,E2 -10983.989} C_VEL
LIN {X 0,Y 404.33,Z 731.727,A -85,B 0,C 180,E1 -10985.986,E2 -10985.986} C_VEL
LIN {X 0,Y 404.377,Z 728.867,A -85,B 0,C 180,E1 -10987.992,E2 -10987.992} C_VEL
LIN {X 0,Y 404.643,Z 724.679,A -85,B 0,C 180,E1 -10990.002,E2 -10990.002} C_VEL
LIN {X 0,Y 404.933,Z 719.072,A -85,B 0,C 180,E1 -10992.021,E2 -10992.021} C_VEL
LIN {X 0,Y 405.494,Z 711.847,A -85,B 0,C 180,E1 -10994.042,E2 -10994.042} C_VEL
LIN {X 0,Y 406.166,Z 704.02,A -85,B 0,C 180,E1 -10995.814,E2 -10995.814} C_VEL
LIN {X 0,Y 406.904,Z 694.491,A -85,B 0,C 180,E1 -10997.593,E2 -10997.593} C_VEL
LIN {X 0,Y 407.665,Z 684.673,A -85,B 0,C 180,E1 -10999.12,E2 -10999.12} C_VEL
LIN {X 0,Y 408.558,Z 672.86,A -85,B 0,C 180,E1 -11000.648,E2 -11000.648} C_VEL
LIN {X 0,Y 409.373,Z 661.501,A -85,B 0,C 180,E1 -11001.875,E2 -11001.875} C_VEL
LIN {X 0,Y 410.074,Z 649.681,A -85,B 0,C 180,E1 -11002.948,E2 -11002.948} C_VEL
LIN {X 0,Y 410.826,Z 635.826,A -85,B 0,C 180,E1 -11003.972,E2 -11003.972} C_VEL
LIN {X 0,Y 411.44,Z 621.277,A -85,B 0,C 180,E1 -11004.819,E2 -11004.819} C_VEL
LIN {X 0,Y 411.846,Z 605.804,A -85,B 0,C 180,E1 -11005.497,E2 -11005.497} C_VEL
LIN {X 0,Y 412.017,Z 589.888,A -85,B 0,C 180,E1 -11005.975,E2 -11005.975} C_VEL
LIN {X 0,Y 412.15,Z 571.405,A -85,B 0,C 180,E1 -11006.368,E2 -11006.368} C_VEL
LIN {X 0,Y 404.337,Z 550.647,A -85,B 0,C 180,E1 -11007.159,E2 -11007.159} C_VEL
LIN {X 0,Y 404.25,Z 550.129,A -85,B 0,C 180,E1 -11007.188,E2 -11007.188} C_VEL
LIN {X 0,Y 404.147,Z 550.143,A -85,B 0,C 180,E1 -11010.284,E2 -11010.284} C_VEL
LIN {X 0,Y 404.146,Z 550.142,A -85,B 0,C 180,E1 -11013.812,E2 -11013.812} C_VEL
LIN {X 0,Y 404.137,Z 550.14,A -85,B 0,C 180,E1 -11016.874,E2 -11016.874} C_VEL
LIN {X 0,Y 404.148,Z 550.144,A -85,B 0,C 180,E1 -11020.079,E2 -11020.079} C_VEL
LIN {X 0,Y 404.153,Z 550.138,A -85,B 0,C 180,E1 -11023.083,E2 -11023.083} C_VEL
LIN {X 0,Y 404.148,Z 550.141,A -85,B 0,C 180,E1 -11025.925,E2 -11025.925} C_VEL
LIN {X 0,Y 404.119,Z 550.146,A -85,B 0,C 180,E1 -11028.634,E2 -11028.634} C_VEL
LIN {X 0,Y 404.158,Z 550.137,A -85,B 0,C 180,E1 -11031.491,E2 -11031.491} C_VEL
LIN {X 0,Y 404.185,Z 550.136,A -85,B 0,C 180,E1 -11034.983,E2 -11034.983} C_VEL
LIN {X 0,Y 404.142,Z 550.147,A -85,B 0,C 180,E1 -11038.553,E2 -11038.553} C_VEL
LIN {X 0,Y 404.194,Z 550.133,A -85,B 0,C 180,E1 -11042,E2 -11042} C_VEL
LIN {X 0,Y 404.176,Z 550.135,A -85,B 0,C 180,E1 -11045.334,E2 -11045.334} C_VEL
LIN {X 0,Y 404.138,Z 550.145,A -85,B 0,C 180,E1 -11048.58,E2 -11048.58} C_VEL
LIN {X 0,Y 404.209,Z 550.13,A -85,B 0,C 180,E1 -11051.761,E2 -11051.761} C_VEL
LIN {X 0,Y 404.205,Z 550.139,A -85,B 0,C 180,E1 -11054.881,E2 -11054.881} C_VEL
LIN {X 0,Y 404.255,Z 550.125,A -85,B 0,C 180,E1 -11057.958,E2 -11057.958} C_VEL
LIN {X 0,Y 404.431,Z 550.103,A -85,B 0,C 180,E1 -11062.099,E2 -11062.099} C_VEL
LIN {X 0,Y 404.422,Z 550.104,A -85,B 0,C 180,E1 -11064.014,E2 -11064.014} C_VEL
LIN {X 0,Y 404.481,Z 550.097,A -85,B 0,C 180,E1 -11068.008,E2 -11068.008} C_VEL
LIN {X 0,Y 404.609,Z 550.081,A -85,B 0,C 180,E1 -11069.999,E2 -11069.999} C_VEL
LIN {X 0,Y 404.422,Z 550.109,A -85,B 0,C 180,E1 -11072.988,E2 -11072.988} C_VEL
LIN {X 0,Y 404.404,Z 550.11,A -85,B 0,C 180,E1 -11076.987,E2 -11076.987} C_VEL
LIN {X 0,Y 404.26,Z 550.125,A -85,B 0,C 180,E1 -11080.011,E2 -11080.011} C_VEL
LIN {X 0,Y 404.257,Z 550.124,A -85,B 0,C 180,E1 -11082.485,E2 -11082.485} C_VEL
LIN {X 0,Y 403.588,Z 550.215,A -85,B 0,C 180,E1 -11083.317,E2 -11083.317} C_VEL
LIN {X 0,Y 400.702,Z 550.568,A -85,B 0,C 180,E1 -11084.668,E2 -11084.668} C_VEL
LIN {X 0,Y 398.267,Z 550.874,A -85,B 0,C 180,E1 -11085.76,E2 -11085.76} C_VEL
LIN {X 0,Y 397.239,Z 550.999,A -85,B 0,C 180,E1 -11086.604,E2 -11086.604} C_VEL
LIN {X 0,Y 397.165,Z 551.009,A -85,B 0,C 180,E1 -11086.89,E2 -11086.89} C_VEL
LIN {X 0,Y 397.134,Z 551.012,A -85,B 0,C 180,E1 -11090.295,E2 -11090.295} C_VEL
LIN {X 0,Y 397.129,Z 551.015,A -85,B 0,C 180,E1 -11094.018,E2 -11094.018} C_VEL
LIN {X 0,Y 397.19,Z 551.009,A -85,B 0,C 180,E1 -11097.39,E2 -11097.39} C_VEL
LIN {X 0,Y 397.087,Z 551.018,A -85,B 0,C 180,E1 -11100.881,E2 -11100.881} C_VEL
LIN {X 0,Y 397.121,Z 551.014,A -85,B 0,C 180,E1 -11104.493,E2 -11104.493} C_VEL
LIN {X 0,Y 397.104,Z 551.018,A -85,B 0,C 180,E1 -11108.274,E2 -11108.274} C_VEL
LIN {X 0,Y 397.107,Z 551.015,A -85,B 0,C 180,E1 -11110.905,E2 -11110.905} C_VEL
LIN {X 0,Y 397.099,Z 551.02,A -85,B 0,C 180,E1 -11113.648,E2 -11113.648} C_VEL
LIN {X 0,Y 397.159,Z 551.01,A -85,B 0,C 180,E1 -11116.511,E2 -11116.511} C_VEL
LIN {X 0,Y 397.119,Z 551.016,A -85,B 0,C 180,E1 -11119.55,E2 -11119.55} C_VEL
LIN {X 0,Y 397.094,Z 551.018,A -85,B 0,C 180,E1 -11122.79,E2 -11122.79} C_VEL
LIN {X 0,Y 397.148,Z 551.01,A -85,B 0,C 180,E1 -11125.115,E2 -11125.115} C_VEL
LIN {X 0,Y 401.852,Z 563.986,A -85,B 0,C 180,E1 -11125.627,E2 -11125.627} C_VEL
LIN {X 0,Y 404.165,Z 570.1,A -85,B 0,C 180,E1 -11125.857,E2 -11125.857} C_VEL
LIN {X 0,Y 403.65,Z 611.828,A -85,B 0,C 180,E1 -11126.733,E2 -11126.733} C_VEL
LIN {X 0,Y 403.468,Z 626.314,A -85,B 0,C 180,E1 -11127.244,E2 -11127.244} C_VEL
LIN {X 0,Y 402.995,Z 640.128,A -85,B 0,C 180,E1 -11127.94,E2 -11127.94} C_VEL
LIN {X 0,Y 402.338,Z 653.87,A -85,B 0,C 180,E1 -11128.861,E2 -11128.861} C_VEL
LIN {X 0,Y 401.659,Z 666.565,A -85,B 0,C 180,E1 -11129.943,E2 -11129.943} C_VEL
LIN {X 0,Y 400.861,Z 677.945,A -85,B 0,C 180,E1 -11131.136,E2 -11131.136} C_VEL
LIN {X 0,Y 400.073,Z 688.855,A -85,B 0,C 180,E1 -11132.541,E2 -11132.541} C_VEL
LIN {X 0,Y 399.443,Z 697.652,A -85,B 0,C 180,E1 -11133.905,E2 -11133.905} C_VEL
LIN {X 0,Y 398.727,Z 706.344,A -85,B 0,C 180,E1 -11135.531,E2 -11135.531} C_VEL
LIN {X 0,Y 398.192,Z 713.448,A -85,B 0,C 180,E1 -11137.152,E2 -11137.152} C_VEL
LIN {X 0,Y 397.734,Z 719.216,A -85,B 0,C 180,E1 -11138.763,E2 -11138.763} C_VEL
LIN {X 0,Y 397.438,Z 723.83,A -85,B 0,C 180,E1 -11140.368,E2 -11140.368} C_VEL
LIN {X 0,Y 397.196,Z 727.426,A -85,B 0,C 180,E1 -11141.963,E2 -11141.963} C_VEL
LIN {X 0,Y 397.017,Z 730.068,A -85,B 0,C 180,E1 -11143.547,E2 -11143.547} C_VEL
LIN {X 0,Y 396.964,Z 731.342,A -85,B 0,C 180,E1 -11144.6,E2 -11144.6} C_VEL
LIN {X 0,Y 396.994,Z 732.727,A -85,B 0,C 180,E1 -11146.695,E2 -11146.695} C_VEL
LIN {X 0,Y 397.08,Z 732.686,A -85,B 0,C 180,E1 -11148.774,E2 -11148.774} C_VEL
LIN {X 0,Y 397.311,Z 731.227,A -85,B 0,C 180,E1 -11150.84,E2 -11150.84} C_VEL
LIN {X 0,Y 397.684,Z 728.298,A -85,B 0,C 180,E1 -11152.894,E2 -11152.894} C_VEL
LIN {X 0,Y 398.207,Z 723.823,A -85,B 0,C 180,E1 -11154.938,E2 -11154.938} C_VEL
LIN {X 0,Y 398.665,Z 719.413,A -85,B 0,C 180,E1 -11156.463,E2 -11156.463} C_VEL
LIN {X 0,Y 399.439,Z 712.901,A -85,B 0,C 180,E1 -11158.236,E2 -11158.236} C_VEL
LIN {X 0,Y 400.253,Z 704.784,A -85,B 0,C 180,E1 -11160,E2 -11160} C_VEL
LIN {X 0,Y 401.183,Z 696.178,A -85,B 0,C 180,E1 -11161.506,E2 -11161.506} C_VEL
LIN {X 0,Y 402.068,Z 685.708,A -85,B 0,C 180,E1 -11163.006,E2 -11163.006} C_VEL
LIN {X 0,Y 403.036,Z 674.976,A -85,B 0,C 180,E1 -11164.251,E2 -11164.251} C_VEL
LIN {X 0,Y 403.832,Z 663.185,A -85,B 0,C 180,E1 -11165.368,E2 -11165.368} C_VEL
LIN {X 0,Y 404.503,Z 651.727,A -85,B 0,C 180,E1 -11166.234,E2 -11166.234} C_VEL
LIN {X 0,Y 404.939,Z 639.341,A -85,B 0,C 180,E1 -11166.979,E2 -11166.979} C_VEL
LIN {X 0,Y 405.266,Z 625.225,A -85,B 0,C 180,E1 -11167.595,E2 -11167.595} C_VEL
LIN {X 0,Y 405.305,Z 610.696,A -85,B 0,C 180,E1 -11168.012,E2 -11168.012} C_VEL
LIN {X 0,Y 405.874,Z 570.486,A -85,B 0,C 180,E1 -11168.824,E2 -11168.824} C_VEL
LIN {X 0,Y 400.862,Z 559.115,A -85,B 0,C 180,E1 -11169.431,E2 -11169.431} C_VEL
LIN {X 0,Y 397.399,Z 551.87,A -85,B 0,C 180,E1 -11169.857,E2 -11169.857} C_VEL
LIN {X 0,Y 397.251,Z 551.004,A -85,B 0,C 180,E1 -11169.91,E2 -11169.91} C_VEL
LIN {X 0,Y 397.223,Z 551.01,A -85,B 0,C 180,E1 -11173.322,E2 -11173.322} C_VEL
LIN {X 0,Y 397.178,Z 551.015,A -85,B 0,C 180,E1 -11177.156,E2 -11177.156} C_VEL
LIN {X 0,Y 397.1,Z 551.021,A -85,B 0,C 180,E1 -11180.731,E2 -11180.731} C_VEL
LIN {X 0,Y 397.13,Z 551.016,A -85,B 0,C 180,E1 -11184.019,E2 -11184.019} C_VEL
LIN {X 0,Y 397.192,Z 551.005,A -85,B 0,C 180,E1 -11187.391,E2 -11187.391} C_VEL
LIN {X 0,Y 397.083,Z 551.016,A -85,B 0,C 180,E1 -11190.883,E2 -11190.883} C_VEL
LIN {X 0,Y 397.123,Z 551.009,A -85,B 0,C 180,E1 -11194.494,E2 -11194.494} C_VEL
LIN {X 0,Y 397.105,Z 551.016,A -85,B 0,C 180,E1 -11198.275,E2 -11198.275} C_VEL
LIN {X 0,Y 397.089,Z 551.022,A -85,B 0,C 180,E1 -11200.909,E2 -11200.909} C_VEL
LIN {X 0,Y 397.102,Z 551.019,A -85,B 0,C 180,E1 -11203.649,E2 -11203.649} C_VEL
LIN {X 0,Y 397.101,Z 551.018,A -85,B 0,C 180,E1 -11206.522,E2 -11206.522} C_VEL
LIN {X 0,Y 397.114,Z 551.018,A -85,B 0,C 180,E1 -11210.424,E2 -11210.424} C_VEL
LIN {X 0,Y 397.134,Z 551.067,A -85,B 0,C 180,E1 -11212.729,E2 -11212.729} C_VEL
LIN {X 0,Y 400.153,Z 565.275,A -85,B 0,C 180,E1 -11216.109,E2 -11216.109} C_VEL
LIN {X 0,Y 401.807,Z 573.789,A -85,B 0,C 180,E1 -11218.056,E2 -11218.056} C_VEL
LIN {X 0,Y 400.507,Z 589.391,A -85,B 0,C 180,E1 -11221.33,E2 -11221.33} C_VEL
LIN {X 0,Y 399.084,Z 608.484,A -85,B 0,C 180,E1 -11225.277,E2 -11225.277} C_VEL
LIN {X 0,Y 397.994,Z 627.57,A -85,B 0,C 180,E1 -11229.167,E2 -11229.167} C_VEL
LIN {X 0,Y 403.687,Z 675.717,A -85,B 0,C 180,E1 -11230.656,E2 -11230.656} C_VEL
LIN {X 0,Y 401.887,Z 742.635,A -85,B 0,C 180,E1 -11232.279,E2 -11232.279} C_VEL
LIN {X 0,Y 401.216,Z 756.327,A -85,B 0,C 180,E1 -11232.807,E2 -11232.807} C_VEL
LIN {X 0,Y 400.354,Z 769.039,A -85,B 0,C 180,E1 -11233.492,E2 -11233.492} C_VEL
LIN {X 0,Y 399.458,Z 780.562,A -85,B 0,C 180,E1 -11234.306,E2 -11234.306} C_VEL
LIN {X 0,Y 398.637,Z 791.953,A -85,B 0,C 180,E1 -11235.32,E2 -11235.32} C_VEL
LIN {X 0,Y 397.799,Z 802.57,A -85,B 0,C 180,E1 -11236.482,E2 -11236.482} C_VEL
LIN {X 0,Y 397.374,Z 810.204,A -85,B 0,C 180,E1 -11237.488,E2 -11237.488} C_VEL
LIN {X 0,Y 396.887,Z 818.433,A -85,B 0,C 180,E1 -11238.768,E2 -11238.768} C_VEL
LIN {X 0,Y 396.531,Z 826.566,A -85,B 0,C 180,E1 -11240.307,E2 -11240.307} C_VEL
LIN {X 0,Y 396.357,Z 833.077,A -85,B 0,C 180,E1 -11241.846,E2 -11241.846} C_VEL
LIN {X 0,Y 396.331,Z 837.816,A -85,B 0,C 180,E1 -11243.234,E2 -11243.234} C_VEL
LIN {X 0,Y 396.454,Z 842.215,A -85,B 0,C 180,E1 -11244.915,E2 -11244.915} C_VEL
LIN {X 0,Y 396.539,Z 844.225,A -85,B 0,C 180,E1 -11245.935,E2 -11245.935} C_VEL
LIN {X 0,Y 396.511,Z 845.761,A -85,B 0,C 180,E1 -11246.953,E2 -11246.953} C_VEL
LIN {X 0,Y 396.527,Z 846.843,A -85,B 0,C 180,E1 -11247.969,E2 -11247.969} C_VEL
LIN {X 0,Y 396.561,Z 847.435,A -85,B 0,C 180,E1 -11248.985,E2 -11248.985} C_VEL
LIN {X 0,Y 396.8,Z 847.622,A -85,B 0,C 180,E1 -11250.001,E2 -11250.001} C_VEL
LIN {X 0,Y 396.575,Z 847.304,A -85,B 0,C 180,E1 -11251.016,E2 -11251.016} C_VEL
LIN {X 0,Y 396.554,Z 846.571,A -85,B 0,C 180,E1 -11252.032,E2 -11252.032} C_VEL
LIN {X 0,Y 396.546,Z 845.355,A -85,B 0,C 180,E1 -11253.048,E2 -11253.048} C_VEL
LIN {X 0,Y 396.552,Z 842.7,A -85,B 0,C 180,E1 -11254.575,E2 -11254.575} C_VEL
LIN {X 0,Y 396.414,Z 837.654,A -85,B 0,C 180,E1 -11256.541,E2 -11256.541} C_VEL
LIN {X 0,Y 396.397,Z 832.087,A -85,B 0,C 180,E1 -11258.155,E2 -11258.155} C_VEL
LIN {X 0,Y 396.504,Z 825.428,A -85,B 0,C 180,E1 -11259.695,E2 -11259.695} C_VEL
LIN {X 0,Y 396.869,Z 817.253,A -85,B 0,C 180,E1 -11261.233,E2 -11261.233} C_VEL
LIN {X 0,Y 397.416,Z 807.192,A -85,B 0,C 180,E1 -11262.771,E2 -11262.771} C_VEL
LIN {X 0,Y 397.737,Z 800.668,A -85,B 0,C 180,E1 -11263.626,E2 -11263.626} C_VEL
LIN {X 0,Y 398.439,Z 791.211,A -85,B 0,C 180,E1 -11264.689,E2 -11264.689} C_VEL
LIN {X 0,Y 399.572,Z 778.885,A -85,B 0,C 180,E1 -11265.821,E2 -11265.821} C_VEL
LIN {X 0,Y 400.696,Z 765.271,A -85,B 0,C 180,E1 -11266.823,E2 -11266.823} C_VEL
LIN {X 0,Y 401.812,Z 752.177,A -85,B 0,C 180,E1 -11267.561,E2 -11267.561} C_VEL
LIN {X 0,Y 402.75,Z 737.47,A -85,B 0,C 180,E1 -11268.175,E2 -11268.175} C_VEL
LIN {X 0,Y 403.262,Z 722.216,A -85,B 0,C 180,E1 -11268.612,E2 -11268.612} C_VEL
LIN {X 0,Y 404.457,Z 673.916,A -85,B 0,C 180,E1 -11269.745,E2 -11269.745} C_VEL
LIN {X 0,Y 402.202,Z 638.723,A -85,B 0,C 180,E1 -11270.836,E2 -11270.836} C_VEL
LIN {X 0,Y 399.729,Z 618.101,A -85,B 0,C 180,E1 -11271.599,E2 -11271.599} C_VEL
LIN {X 0,Y 397.421,Z 603.954,A -85,B 0,C 180,E1 -11272.21,E2 -11272.21} C_VEL
LIN {X 0,Y 397.821,Z 587.24,A -85,B 0,C 180,E1 -11275.405,E2 -11275.405} C_VEL
LIN {X 0,Y 398.384,Z 570.32,A -85,B 0,C 180,E1 -11278.733,E2 -11278.733} C_VEL
LIN {X 0,Y 398.757,Z 560.443,A -85,B 0,C 180,E1 -11280.739,E2 -11280.739} C_VEL
LIN {X 0,Y 397.193,Z 551.014,A -85,B 0,C 180,E1 -11282.831,E2 -11282.831} C_VEL
LIN {X 0,Y 397.113,Z 551.018,A -85,B 0,C 180,E1 -11285.735,E2 -11285.735} C_VEL
LIN {X 0,Y 397.118,Z 551.016,A -85,B 0,C 180,E1 -11289.577,E2 -11289.577} C_VEL
LIN {X 0,Y 397.106,Z 551.018,A -85,B 0,C 180,E1 -11293.479,E2 -11293.479} C_VEL
LIN {X 0,Y 397.107,Z 551.018,A -85,B 0,C 180,E1 -11296.521,E2 -11296.521} C_VEL
LIN {X 0,Y 397.119,Z 551.017,A -85,B 0,C 180,E1 -11300.423,E2 -11300.423} C_VEL
LIN {X 0,Y 397.112,Z 551.018,A -85,B 0,C 180,E1 -11304.265,E2 -11304.265} C_VEL
LIN {X 0,Y 397.119,Z 551.019,A -85,B 0,C 180,E1 -11306.727,E2 -11306.727} C_VEL
LIN {X 0,Y 397.129,Z 551.019,A -85,B 0,C 180,E1 -11310.296,E2 -11310.296} C_VEL
LIN {X 0,Y 397.199,Z 551.011,A -85,B 0,C 180,E1 -11312.61,E2 -11312.61} C_VEL
LIN {X 0,Y 397.138,Z 551.019,A -85,B 0,C 180,E1 -11315.982,E2 -11315.982} C_VEL
LIN {X 0,Y 397.153,Z 551.018,A -85,B 0,C 180,E1 -11317.468,E2 -11317.468} C_VEL
LIN {X 0,Y 398.221,Z 553.972,A -85,B 0,C 180,E1 -11317.627,E2 -11317.627} C_VEL
LIN {X 0,Y 403.777,Z 564.714,A -85,B 0,C 180,E1 -11318.328,E2 -11318.328} C_VEL
